	91:
		bTimer1															:= TRUE;
		IF tonTimer1.Q THEN
			bTimer1														:= FALSE;
			i4Step														:= 99;
		END_IF
		
	98:																														// Utility error hold - cleared by P_M01
		i4Step															:= 98;
		
	99:
		bRepressurizationDone											:= TRUE;
//		IF NOT bMultiProcess THEN
		Steam_Service_Req												:= FALSE;
//		END_IF
		Current_Step													:= 0;
		i4Step															:= 0;
	
END_CASE

IF i4Step > 0 AND i4Step < 80 THEN
	IF bMultiProcess THEN
		IF U.safe_shutdown_error_1 <> '' AND giSafeShutdown1RS = 0 THEN
			sSafeShutdownError1											:= U.safe_shutdown_error_1;
			giSafeShutdown1RS											:= RS_Number;
		ELSIF U.safe_shutdown_error_2 <> '' AND giSafeShutdown23RS = 0 THEN
			sSafeShutdownError2											:= U.safe_shutdown_error_2;
			giSafeShutdown23RS											:= RS_Number;
		ELSIF (giEvacuationErrorRS + giDesorptionErrorRS + giSafeShutdown1RS + giSafeShutdown23RS) > 0 THEN
			Cancel_Reactor_Set											:= TRUE;
		ELSIF U.os_air_unsafe_temp THEN
			Stop_Reactor_Set											:= TRUE;
		END_IF
	END_IF
	iStep																:= i4Step;
	Current_Step														:= iStep;
	A_Check_Process();
	i4Step																:= iStep;
END_IF
END_ACTION

ACTION A5_Adsorption:
// Phase 0 - FB_Reactor_Set.A5_Adsorption
// Rev 1.0 - May 13, 2024

CASE i5Step OF
	
	0:	;
		
	1:
		Cycle_Stage														:= 'adsorption.initialize';							// 2.d
		iRestartStep													:= 1;
		rTime2															:= m01.SP_adsorption_duration;						// 12
		IF R_S.reactor_pressure_error <> '' THEN
			sReactorError												:= R_S.reactor_pressure_error;
			sMessage													:= gsProcessCannotRun;
		ELSIF R_S.inlet_air_high_temp_count > _INLET_AIR_MAX_COUNT THEN
			sReactorError												:= F_Concat3(INT_TO_STRING(R_S.inlet_air_high_temp_count), ' ', gsSorbentTemperatureError);
			sMessage													:= gsProcessCannotRun;
		ELSE
			i5Step														:= i5Step + 1;
		END_IF
			
	2:
		IF NOT bMultiProcess THEN
			IF R_S.average_reactor_pressure_within_ambient THEN																// 2.c
				sReactorError											:= gsReactorsAtAmbientPressure;
				sMessage												:= gsProcessComplete;
			ELSIF NOT R_S.all_clamps_retracted THEN																			// 2.a
				sReactorError											:= gsDoorClampsExtendedError;
				sMessage												:= gsProcessCannotRun;
			ELSIF u.os_air_unsafe_temp THEN																					// 2.b
				sReactorError											:= gsOutsideTempRangeError;
				sMessage												:= gsProcessCannotRun;
			ELSE
				i5Step													:= i5Step + 1;
			END_IF
		ELSE
			i5Step														:= i5Step + 1;
		END_IF

	3:
		bTimer2															:= TRUE;											// 4
		IF R_S.r1_inlet_co2 < m01.SP_minimum_desired_inlet_co2_concentration_during_adsorption THEN							// 5.a
			sError														:= gsAdsorptionInletCo2LowError;
			sMessage													:= gsAdsorptionCo2LowCheck;
		END_IF
		R_S.close_all_valves											:= TRUE;											// 5.b
		U.drainage_on													:= TRUE;											// 5.d
		R_S.fan_vfd_percent												:= 0;												// 5.e
		rTime1															:= _VALVE_TIME;
		i5Step															:= i5Step + 1;
		
	4:
		bTimer1															:= TRUE;
		IF R_S.valves_clear THEN
			bTimer1														:= FALSE;
			i5Step														:= i5Step + 1;
		ELSIF tonTimer1.Q THEN
			bTimer1														:= FALSE;
			sReactorError												:= SEL(R_S.steam_control_valve_closed, gsSteamControlValveError, '');
			sReactorError												:= SEL(R_S.dead_air_valve_clear, gsDeadAirValveError, sReactorError);
			sReactorError												:= SEL(R_S.purge_valve_clear, gsPurgeValveError, sReactorError);
			sReactorError												:= SEL(R_S.cooling_valve_clear, gsCoolingValveError, sReactorError);
			sReactorError												:= SEL(R_S.steam_header_valve_clear, gsSteamHeaderValveError, sReactorError);
			sMessage													:= gsReactorSetCannotRun;
		END_IF

	5:
		R_S.open_repres_valves											:= TRUE;											// 6
		rTime1															:= _VALVE_TIME;
		i5Step															:= i5Step + 1;

	6:
		bTimer1															:= TRUE;
		IF R_S.repres_valve_error = '' THEN
			bTimer1														:= FALSE;
			R_S.co2_outside_sensors_on									:= TRUE;											// 7
			R_S.open_all_doors											:= TRUE;											// 8
			Cycle_Stage													:= 'adsorption.open_doors';							// 8.a
			rTime1														:= m01.SP_doorsopenclose_timedelay * _MINUTES;		// 8.b
			i5Step														:= i5Step + 1;
		ELSIF tonTimer1.Q THEN
			bTimer1														:= FALSE;
			sReactorError												:= R_S.repres_valve_error;
			sMessage													:= gsProcessCannotRun;
		END_IF
							
	7:
		bTimer1															:= TRUE;
		IF R_S.all_doors_open THEN
			bTimer1														:= FALSE;
			R_S.fan_vfd_percent											:= Fan_setpoint;									// 9
			Cycle_Stage													:= 'adsorption.turn_on_fans';						// 9.a
			rSP1														:= m01.SP_unacceptable_duration_from_adsorption_start_until_sorbent_cool * _MINUTES;	// 10.c
			rSP2														:= m01.SP_undesirable_duration_from_adsorption_start_until_sorbent_cool * _MINUTES;		// 10.b
			rSP3														:= m01.SP_target_duration_from_adsorption_start_until_sorbent_cool * _MINUTES;			// 10.a
			i5Step														:= i5Step + 1;
		ELSIF tonTimer1.Q THEN
			bTimer1														:= FALSE;
			sReactorError												:= gsDoorsNotOpenError;
			sMessage													:= gsProcessCannotRun;
		END_IF
		
	8:
		rTime															:= TIME_TO_REAL(tonTimer2.ET);
		IF rTime >= rSP1 THEN																								// 10.c
			IF R_S.inlet_air_high_temp_count = 0 THEN																		// 10.c.i
				sPauseError												:= gsAdsorptionUnacceptableTimeError;
				sMessage												:= gsReactorSetWillPause;												
			ELSE
				sSafeShutdownError1										:= gsAdsorptionTimeOutError;						// 10.c.ii - Safe Shutdown 1
			END_IF
		ELSIF rTime >= rSP2 THEN																							// 10.b
			IF R_S.inlet_air_high_temp_count = 0 THEN
				sError													:= gsAdsorptionAcceptableButNotIdealTimeError;																
				i5Step													:= i5Step + 1;
			END_IF
		ELSIF rTime >= rSP3 THEN																							// 10.c
			IF R_S.inlet_air_high_temp_count = 0 THEN																	
				i5Step													:= i5Step + 1;
			END_IF
		END_IF

	9:
		R_S.co2_inside_sensors_on										:= TRUE;											// 11
		Cycle_Stage														:= 'adsorption.adsorption';							// 11.a
		i5Step 															:= i5Step + 1;
		
	10:
		IF tonTimer2.Q THEN																									// 12
			bTimer2														:= FALSE;
			R_S.fan_vfd_percent											:= 0;
			Cycle_Stage													:= 'adsorption.turn_off_fans';						// 12.a
			rTime1														:= _FAN_SHUTDOWN_TIME;
			i5Step														:= i5Step + 1;
		END_IF

	11:
		bTimer1															:= TRUE;
		IF tonTimer1.Q THEN
			bTimer1														:= FALSE;	
			R_S.close_all_doors											:= TRUE;											// 13
			Cycle_Stage													:= 'adsorption.close_doors';						// 13.a
			rTime1														:= m01.SP_doorsopenclose_timedelay * _MINUTES;										// 13.b
			i5Step														:= i5Step + 1;
		END_IF
		
	12:
		bTimer1															:= TRUE;
		IF tonTimer1.Q THEN
			bTimer1														:= FALSE;
			R_S.co2_sensors_off											:= TRUE;											// 14
			rTime1														:= m01.SP_dead_time_in_cycle_duration;				// 15
			Cycle_Stage													:= 'adsorption.cycle_dead_time';					// 15.a
			i5Step														:= i5Step + 1;
		END_IF
		
	13:
		bTimer1															:= TRUE;
		IF tonTimer1.Q THEN
			bTimer1														:= FALSE;
			i5Step														:= 99;
		END_IF
				
	80:																														// Manual process closing
		Cycle_Stage														:= 'adsorption.stopping';
		R_S.fan_vfd_percent												:= 0;
		R_S.co2_sensors_off												:= TRUE;
		R_S.close_repres_valves											:= TRUE;
		rTime1															:= _STOPPING_TIME;
		i5Step															:= i5Step + 1;
		
	81:
		bTimer1															:= TRUE;
		IF tonTimer1.Q THEN
			bTimer1														:= FALSE;
			i5Step														:= 99;
		END_IF
		
	90:																														// Automatic process stopping
		Cycle_Stage														:= 'adsorption.stopping';
		R_S.fan_vfd_percent												:= 0;
		R_S.co2_sensors_off												:= TRUE;
		R_S.close_repres_valves											:= TRUE;
		rTime1															:= _STOPPING_TIME;
		i5Step															:= i5Step + 1;
		
	91:
		bTimer1															:= TRUE;
		IF tonTimer1.Q THEN
			bTimer1														:= FALSE;
			i5Step														:= 99;
		END_IF
		
	98:																														// Utility error hold - cleared by P_M01
		i5Step															:= 98;
		
	99:
		bAdsorptionDone													:= TRUE;
		bTimer2															:= FALSE;
		U.drainage_on													:= FALSE;
		Current_Step													:= 0;
		i5Step															:= 0;
	
END_CASE

IF i5Step > 0 AND i5Step < 80 THEN
	IF bMultiProcess THEN
		IF U.safe_shutdown_error_1 <> '' AND giSafeShutdown1RS = 0 THEN
			sSafeShutdownError1											:= U.safe_shutdown_error_1;
			giSafeShutdown1RS											:= RS_Number;
		ELSIF U.safe_shutdown_error_2 <> '' AND giSafeShutdown23RS = 0 THEN
			sSafeShutdownError2											:= U.safe_shutdown_error_2;
			giSafeShutdown23RS											:= RS_Number;
		ELSIF sSafeShutdownError1 <> '' AND giSafeShutdown1RS = 0 THEN
			giSafeShutdown1RS											:= RS_Number;
		ELSIF (giEvacuationErrorRS + giDesorptionErrorRS + giSafeShutdown1RS + giSafeShutdown23RS) > 0 THEN
			Cancel_Reactor_Set											:= TRUE;
		ELSIF U.os_air_unsafe_temp THEN
			Stop_Reactor_Set											:= TRUE;
		END_IF
	END_IF
	iStep																:= i5Step;
	Current_Step														:= iStep;
	A_Check_Process();
	i5Step																:= iStep;
END_IF
END_ACTION

ACTION A5_Adsorption_Test:
// Phase 0 - FB_Reactor_Set.A5_Adsorption_Test
// Rev 1.0 - June 3, 2024

CASE i5Step OF	

	0:	;
		
	1:
		Cycle_Stage														:= 'adsorption.initialize';							// 2.d
		//iRestartStep													:= 1;
		rTime2															:= m01.SP_adsorption_duration * _MINUTES;			// 12
		IF R_S.reactor_pressure_error <> '' THEN
			sReactorError												:= R_S.reactor_pressure_error;
			sMessage													:= gsProcessCannotRun;
		ELSE
			R_S.retract_all_clamps 										:= TRUE;
			rTime1														:= m01.SP_clampsretract_timedelay;
			i5Step														:= i5Step + 1;
		END_IF
			
	2:
		IF NOT bMultiProcess THEN
			IF R_S.average_reactor_pressure_within_ambient THEN																// 2.c
				sReactorError											:= gsReactorsAtAmbientPressure;
				sMessage												:= gsProcessComplete;
			ELSE
				i5Step													:= i5Step + 1;
			END_IF
		ELSE
			i5Step														:= i5Step + 1;
		END_IF

	3:
		bTimer1															:= TRUE;
		IF R_S.all_clamps_retracted THEN																					// 2.a
			bTimer1														:= FALSE;
			i5Step														:= i5Step + 1;
		ELSE
			sReactorError												:= gsDoorClampsExtendedError;
			sMessage													:= gsProcessCannotRun;
		END_IF
		
	4:
		R_S.close_all_valves											:= TRUE;											// 5.b
		U.drainage_on													:= TRUE;											// 5.d
		R_S.fan_vfd_percent												:= 0;												// 5.e
		rTime1															:= _VALVE_TIME;
		i5Step															:= i5Step + 1;
		
	5:
		bTimer1															:= TRUE;
		IF R_S.valves_clear THEN
			bTimer1														:= FALSE;
			i5Step														:= i5Step + 2;
		ELSIF tonTimer1.Q THEN
			bTimer1														:= FALSE;
			sReactorError												:= SEL(R_S.steam_control_valve_closed, gsSteamControlValveError, '');
			sReactorError												:= SEL(R_S.dead_air_valve_clear, gsDeadAirValveError, sReactorError);
			sReactorError												:= SEL(R_S.purge_valve_clear, gsPurgeValveError, sReactorError);
			sReactorError												:= SEL(R_S.cooling_valve_clear, gsCoolingValveError, sReactorError);
			sReactorError												:= SEL(R_S.steam_header_valve_clear, gsSteamHeaderValveError, sReactorError);
			sMessage													:= gsReactorSetCannotRun;
		END_IF

	6:
		R_S.open_repres_valves											:= TRUE;											// 6
		rTime1															:= _VALVE_TIME;
		i5Step															:= i5Step + 1;

	7:
		bTimer1															:= TRUE;
		IF R_S.repres_valve_error = '' THEN
			bTimer1														:= FALSE;
			R_S.co2_inside_sensors_on									:= TRUE;											// 7
			R_S.open_all_doors											:= TRUE;											// 8
			Cycle_Stage													:= 'adsorption.open_doors';							// 8.a
			rTime1														:= m01.SP_doorsopenclose_timedelay * _MINUTES;		// 8.b
			i5Step														:= i5Step + 1;
		ELSIF tonTimer1.Q THEN
			bTimer1														:= FALSE;
			sReactorError												:= R_S.repres_valve_error;
			sMessage													:= gsProcessCannotRun;
		END_IF
							
	8:
		bTimer1															:= TRUE;
		//IF R_S.all_doors_open THEN
		IF tonTimer1.Q THEN
			bTimer1														:= FALSE;
			R_S.close_repres_valves										:= TRUE;		
			R_S.fan_vfd_percent											:= Fan_setpoint;									// 9
			Cycle_Stage													:= 'adsorption.turn_on_fans';						// 9.a
		
			i5Step														:= i5Step + 1;
		END_IF
		
	9:
		IF R_S.sorbent_high_temp <=  m01.SP_adsorption_sorbent_hightemp_startco2analyzer THEN 
				i5Step														:= i5Step + 1;
		END_IF

	10:
		//R_S.co2_inside_sensors_on										:= TRUE;											// 11
		bTimer2															:= TRUE;	
		Cycle_Stage														:= 'adsorption.adsorption';							// 11.a
		IF R_S.R1_outlet_co2 >= m01.SP_adsorption_outletco2_highlimit AND tonTimer2.Q THEN
			bTimer2															:= FALSE;	
			i5Step 															:= i5Step + 1;
		END_IF
		
	11:
		
		R_S.fan_vfd_percent											:= 0;
		Cycle_Stage													:= 'adsorption.turn_off_fans';						// 12.a
		rTime1														:= _FAN_SHUTDOWN_TIME;
		i5Step														:= i5Step + 1;
	

	12:
		bTimer1															:= TRUE;
		IF tonTimer1.Q THEN
			bTimer1														:= FALSE;	
			R_S.close_all_doors											:= TRUE;											// 13
			Cycle_Stage													:= 'adsorption.close_doors';						// 13.a
			rTime1														:= m01.SP_doorsopenclose_timedelay * _MINUTES;										// 13.b
			i5Step														:= i5Step + 1;
		END_IF
		
	13:
		bTimer1															:= TRUE;
		IF tonTimer1.Q THEN
			bTimer1														:= FALSE;
			R_S.co2_sensors_off											:= TRUE;											// 14
			rTime1														:= m01.SP_dead_time_in_cycle_duration;				// 15
			Cycle_Stage													:= 'adsorption.cycle_dead_time';					// 15.a
			i5Step														:= i5Step + 1;
		END_IF
		
	14:
		bTimer1															:= TRUE;
		IF tonTimer1.Q THEN
			bTimer1														:= FALSE;
			i5Step														:= 99;
		END_IF
				
	80:																														// Manual process closing
		Cycle_Stage														:= 'adsorption.stopping';
		R_S.fan_vfd_percent												:= 0;
		R_S.co2_sensors_off												:= TRUE;
		R_S.close_repres_valves											:= TRUE;
		rTime1															:= _STOPPING_TIME;
		i5Step															:= i5Step + 1;
		
	81:
		bTimer1															:= TRUE;
		IF tonTimer1.Q THEN
			bTimer1														:= FALSE;
			i5Step														:= 99;
		END_IF
		
	90:																														// Automatic process stopping
		Cycle_Stage														:= 'adsorption.stopping';
		R_S.fan_vfd_percent												:= 0;
		R_S.co2_sensors_off												:= TRUE;
		R_S.close_repres_valves											:= TRUE;
		rTime1															:= _STOPPING_TIME;
		i5Step															:= i5Step + 1;
		
	91:
		bTimer1															:= TRUE;
		IF tonTimer1.Q THEN
			bTimer1														:= FALSE;
			i5Step														:= 99;
		END_IF
		
	98:																														// Utility error hold - cleared by P_M01
		i5Step															:= 98;
		
	99:
		bAdsorptionDone													:= TRUE;
		//bTimer2															:= FALSE;
		U.drainage_on													:= FALSE;
		Current_Step													:= 0;
		i5Step															:= 0;
	
END_CASE

IF i5Step > 0 AND i5Step < 80 THEN
	IF bMultiProcess THEN
		IF U.safe_shutdown_error_1 <> '' AND giSafeShutdown1RS = 0 THEN
			sSafeShutdownError1											:= U.safe_shutdown_error_1;
			giSafeShutdown1RS											:= RS_Number;
		ELSIF U.safe_shutdown_error_2 <> '' AND giSafeShutdown23RS = 0 THEN
			sSafeShutdownError2											:= U.safe_shutdown_error_2;
			giSafeShutdown23RS											:= RS_Number;
		ELSIF sSafeShutdownError1 <> '' AND giSafeShutdown1RS = 0 THEN
			giSafeShutdown1RS											:= RS_Number;
		ELSIF (giEvacuationErrorRS + giDesorptionErrorRS + giSafeShutdown1RS + giSafeShutdown23RS) > 0 THEN
			Cancel_Reactor_Set											:= TRUE;
		ELSIF U.os_air_unsafe_temp THEN
			Stop_Reactor_Set											:= TRUE;
		END_IF
	END_IF
	iStep																:= i5Step;
	Current_Step														:= iStep;
	A_Check_Process();
	i5Step																:= iStep;
END_IF
END_ACTION

ACTION A5_Adsorption_Test_Auto:
// Phase 0 - FB_Reactor_Set.A5_Adsorption_Test
// Rev 1.0 - June 3, 2024

CASE i5Step OF	

	0:	;
		
	1:
		Cycle_Stage														:= 'adsorption.initialize';							// 2.d
		//iRestartStep													:= 1;
		rTime1														:= 5 * _SECONDS;
		i5Step														:= i5Step + 1;
		
			
	2:
		bTimer1 := TRUE;
		IF sita_bits[3].1 THEN 
			bTimer1 := FALSE;
			i5Step := 90;
		ELSIF tonTimer1.Q AND  sita_bits[3].2 THEN 
			bTimer1														:= FALSE;
			sReactorError												:= 'Adsorption Error';
			sMessage													:= 'Auto Test';
		END_IF

	
	80:																														// Manual process closing
		Cycle_Stage														:= 'adsorption.stopping';
		rTime1															:= _STOPPING_TIME;
		i5Step															:= i5Step + 1;
		
	81:
		bTimer1															:= TRUE;
		IF tonTimer1.Q THEN
			bTimer1														:= FALSE;
			i5Step														:= 99;
		END_IF
		
	90:																														// Automatic process stopping
		Cycle_Stage														:= 'adsorption.stopping';
		rTime1															:= _STOPPING_TIME;
		i5Step															:= i5Step + 1;
		
	91:
		bTimer1															:= TRUE;
		IF tonTimer1.Q THEN
			bTimer1														:= FALSE;
			i5Step														:= 99;
		END_IF
		
	98:																														// Utility error hold - cleared by P_M01
		i5Step															:= 98;
		
	99:
		bAdsorptionDone													:= TRUE;
		//bTimer2															:= FALSE;
		U.drainage_on													:= FALSE;
		Current_Step													:= 0;
		i5Step															:= 0;
	
END_CASE

IF i5Step > 0 AND i5Step < 80 THEN
	IF bMultiProcess THEN
		IF U.safe_shutdown_error_1 <> '' AND giSafeShutdown1RS = 0 THEN
			sSafeShutdownError1											:= U.safe_shutdown_error_1;
			giSafeShutdown1RS											:= RS_Number;
		ELSIF U.safe_shutdown_error_2 <> '' AND giSafeShutdown23RS = 0 THEN
			sSafeShutdownError2											:= U.safe_shutdown_error_2;
			giSafeShutdown23RS											:= RS_Number;
		ELSIF sSafeShutdownError1 <> '' AND giSafeShutdown1RS = 0 THEN
			giSafeShutdown1RS											:= RS_Number;
		ELSIF (giEvacuationErrorRS + giDesorptionErrorRS + giSafeShutdown1RS + giSafeShutdown23RS) > 0 THEN
			Cancel_Reactor_Set											:= TRUE;
		ELSIF U.os_air_unsafe_temp THEN
			Stop_Reactor_Set											:= TRUE;
		END_IF
	END_IF
	iStep																:= i5Step;
	Current_Step														:= iStep;
	A_Check_Process();
	i5Step																:= iStep;
END_IF
END_ACTION

ACTION A6_Evacuation:
// Phase 0 - FB_State_Machine.A6_Evacuation
// Rev 1.0 - May 13, 2024

CASE i6Step OF
	
	0:	;
	
	1:
		Cycle_Stage														:= 'evacuation.initialize';							// 1.a
		iRestartStep													:= 1;
		rTime2															:= m01.SP_evacuation_duration;
		IF U.utility_error <> '' THEN																						// 2
			sUtilityError												:= U.utility_error;
			sMessage													:= gsSystemCannotRun;
		ELSIF R_S.reactor_pressure_error <> '' THEN
			sReactorError												:= R_S.reactor_pressure_error;
			sMessage													:= gsReactorSetCannotRun;
		ELSE
			R_S.close_all_doors											:= TRUE;
			rTime1														:= m01.SP_doorsopenclose_timedelay * _MINUTES;
			i6Step														:= i6Step + 1;
		END_IF
		
	2:
		bTimer1															:= TRUE;
		IF R_S.all_doors_closed THEN																						// 1.c.ii
			bTimer1														:= FALSE;
			R_S.close_all_valves										:= TRUE;											// 4.a
			rTime1														:= _VALVE_TIME; 
			i6Step														:= i6Step + 1;
		ELSIF tonTimer1.Q THEN
			bTimer1														:= FALSE;
			sReactorError												:= gsDoorsNotClosedError;
			sMessage													:= gsReactorSetCannotRun;
		END_IF

	3:
		bTimer1															:= TRUE;
		bTimer2															:= TRUE;											// 3
		IF R_S.valves_clear THEN
			bTimer1														:= FALSE;
			U.product_vacuum_backfeed_valve								:= _OPEN;											// 4.a.ii
			rTime1														:= _VALVE_TIME; 
			i6Step														:= i6Step + 1;
		ELSIF tonTimer1.Q THEN
			bTimer1														:= FALSE;
			sReactorError												:= SEL(R_S.steam_control_valve_closed, gsSteamControlValveError, '');
			sReactorError												:= SEL(R_S.dead_air_valve_clear, gsDeadAirValveError, sReactorError);
			sReactorError												:= SEL(R_S.purge_valve_clear, gsPurgeValveError, sReactorError);
			sReactorError												:= SEL(R_S.cooling_valve_clear, gsCoolingValveError, sReactorError);
			sReactorError												:= SEL(R_S.steam_header_valve_clear, gsSteamHeaderValveError, sReactorError);
			sMessage													:= gsReactorSetCannotRun;
		END_IF

	4:
		bTimer1															:= TRUE;
		IF U.product_vacuum_backfeed_valve_open THEN
			bTimer1														:= FALSE;
			U.drainage_on												:= TRUE;											// 4.c
			R_S.co2_outside_sensors_on									:= TRUE;											// 5
			R_S.close_repres_valves										:= TRUE;											// 6
			rTime1														:= _VALVE_TIME; 
			i6Step														:= i6Step + 1;
		ELSIF tonTimer1.Q THEN
			bTimer1														:= FALSE;
			sUtilityError												:= gsProductVacuumBackfeedValveError;
			sMessage													:= gsSystemCannotRun;
		END_IF
			
	5:		
		bTimer1															:= TRUE;	
		IF R_S.repres_valve_error = '' THEN
			bTimer1														:= FALSE;
			R_S.extend_all_clamps										:= TRUE;											// 7
			U.dead_air_vacuum_pump										:= TRUE;											// 8
			Cycle_Stage													:= 'evacuation.evacuate_lines';						// 8.a
			i6Step														:= i6Step + 1;
		ELSIF tonTimer1.Q THEN
			bTimer1														:= FALSE;
			sReactorError												:= R_S.repres_valve_error;
			sMessage													:= gsProcessCannotRun;
		END_IF
		
	6:
		IF U.dead_air_line_pres < m01.SP_evacuation_unacceptable_pressure THEN												// 9
			R_S.dead_air_valve											:= TRUE;											// 9.a
			Cycle_Stage													:= 'evacuation.evacuation';							// 10
			i6Step														:= i6Step + 1;			
		ELSIF tonTimer2.Q OR U.dead_air_line_pres_error THEN																// 9.b
			bTimer2														:= FALSE;
			sReactorError												:= gsUnableToEvacuateLinesError;					// Raise error & stop reactor set				
			sMessage													:= gsSystemWillStop;
			bEvacuationRSError											:= TRUE;											// Stop evacuation for all reactor sets in evacuation. Allow other reactor sets to complete their current cycle.
		END_IF
		 
	7:
		IF tonTimer2.Q THEN																									// 11
			bTimer2														:= FALSE;											// 14
			iStatus														:= F_LowMidHigh(R_S.average_reactor_pressure, m01.SP_evacuation_ideal_pressure, m01.SP_evacuation_unacceptable_pressure, 0);
			IF iStatus = eLow THEN																							// 11.a
				i6Step													:= i6Step + 1;
			ELSIF iStatus = eMid THEN																						// 11.b
				sError													:= gsVacuumPressureAcceptableBotNotIdealError;
				sMessage												:= gsProcessWillContinue;
				i6Step													:= i6Step + 1;
			ELSE																											// 11.c
				sReactorError											:= gsInsufficientVacuumPressureError;
				sMessage												:= gsReactorSetWillPause;
			END_IF
		END_IF
	
	8:
		R_S.dead_air_valve												:= FALSE;											// 12
		U.dead_air_vacuum_pump											:= FALSE;											// 13
		IF R_S.all_clamps_extended THEN																						// 15
			i6Step														:= i6Step + 1;
		ELSE
			sReactorError												:= gsClampExtendError;
			sMessage													:= gsProcessCannotContinue;
		END_IF

	9:
		Cycle_Stage														:= 'evacuation.leak_check';							// 16
		rTime2															:= m01.SP_leak_test_duration;						// 17
		rR1SavedPressure												:= R_S.R1_reactor_pres;
		rR2SavedPressure												:= R_S.R2_reactor_pres;
		rR3SavedPressure												:= R_S.R3_reactor_pres;
		rR4SavedPressure												:= R_S.R4_reactor_pres;
		i6Step															:= i6Step + 1;

	10:
		bTimer2															:= TRUE;
		IF tonTimer2.Q THEN																									// 18
			bTimer2														:= FALSE;
			rR1SavedPressure											:= R_S.R1_reactor_pres - rR1SavedPressure;
			rR2SavedPressure											:= R_S.R2_reactor_pres - rR2SavedPressure;
			rR3SavedPressure											:= R_S.R3_reactor_pres - rR3SavedPressure;
			rR4SavedPressure											:= R_S.R4_reactor_pres - rR4SavedPressure;
			rSP1														:= m01.SP_target_pressure_change;
			rSP2														:= m01.SP_unacceptable_pressure_change;
			iR1Leakage													:= F_LowMidHigh(rR1SavedPressure, rSP1, rSP2, 0);
			iR2Leakage													:= F_LowMidHigh(rR2SavedPressure, rSP1, rSP2, 0);
			iR3Leakage													:= F_LowMidHigh(rR3SavedPressure, rSP1, rSP2, 0);
			iR4Leakage													:= F_LowMidHigh(rR4SavedPressure, rSP1, rSP2, 0);
			sLeakageAcceptable											:= SEL(iR1Leakage = 1, '', 'R1 ');
			sLeakageAcceptable											:= SEL(iR2Leakage = 1, sLeakageAcceptable, CONCAT(sLeakageAcceptable, 'R2 '));
			sLeakageAcceptable											:= SEL(iR3Leakage = 1, sLeakageAcceptable, CONCAT(sLeakageAcceptable, 'R3 '));
			sLeakageAcceptable											:= SEL(iR4Leakage = 1, sLeakageAcceptable, CONCAT(sLeakageAcceptable, 'R4 '));
			sLeakageUnacceptable										:= SEL(iR1Leakage = 2, '', 'R1 ');
			sLeakageUnacceptable										:= SEL(iR2Leakage = 2, sLeakageUnacceptable, CONCAT(sLeakageUnacceptable, 'R2 '));
			sLeakageUnacceptable										:= SEL(iR3Leakage = 2, sLeakageUnacceptable, CONCAT(sLeakageUnacceptable, 'R3 '));
			sLeakageUnacceptable										:= SEL(iR4Leakage = 2, sLeakageUnacceptable, CONCAT(sLeakageUnacceptable, 'R4 '));
			IF sLeakageUnacceptable = '' THEN
				R_S.vacuum_holding										:= TRUE;											// 18.a.i
				R_S.co2_sensors_off										:= TRUE;											// 19
				IF sLeakageAcceptable <> '' THEN
					sError												:= CONCAT(sLeakageAcceptable, gsVacuumPressureAcceptableBotNotIdealError);		// 18.b.i
					sMessage											:= gsReactorSetWillContinue;
				END_IF																										// else 18.a
				i6Step													:= 99;
			ELSE
				R_S.vacuum_holding										:= FALSE;											// 18.c.ii
				sReactorError											:= CONCAT(sLeakageUnacceptable, gsVacuumPressureUnacceptableError);				// 18.c.i
				sMessage												:= gsReactorSetWillPause;
			END_IF
		END_IF			
		
	80:																														// Stop process
		Cycle_Stage														:= 'evacuation.stopping';
		R_S.co2_sensors_off												:= TRUE;
		R_S.dead_air_valve												:= FALSE;
		U.dead_air_vacuum_pump											:= FALSE;
		U.product_vacuum_backfeed_valve									:= _CLOSED;
		rTime1															:= _STOPPING_TIME;
		i6Step															:= i6Step + 1;
		
	81:
		bTimer1															:= TRUE;
		IF tonTimer1.Q THEN
			bTimer1														:= FALSE;
			i6Step														:= 99;
		END_IF

	90:																														// Automatic process stopping
		Cycle_Stage														:= 'evacuation.stopping';
		R_S.co2_sensors_off												:= TRUE;
		R_S.dead_air_valve												:= FALSE;
		U.dead_air_vacuum_pump											:= FALSE;
		U.product_vacuum_backfeed_valve									:= _CLOSED;
		rTime1															:= _STOPPING_TIME;
		i6Step															:= i6Step + 1;
		
	91:
		bTimer1															:= TRUE;
		IF tonTimer1.Q THEN
			bTimer1														:= FALSE;
			i6Step														:= 99;
		END_IF
		
	98:																														// Utility error hold - cleared by P_M01
		i6Step															:= 98;
		
	99:
		IF bStopAfterEvacuation THEN
			bStop														:= TRUE;
			Stop_M01_RS													:= TRUE;											// Stop Reactor in P_M01.A_AutoMode
			bStopAfterEvacuation										:= FALSE;
		END_IF
		bEvacuationDone													:= TRUE;
		U.drainage_on													:= FALSE;
		Current_Step													:= 0;
		i6Step															:= 0;
	
END_CASE

IF i6Step > 0 AND i6Step < 80 THEN
	IF bMultiProcess THEN
		IF U.safe_shutdown_error_1 <> '' AND giSafeShutdown1RS = 0 THEN
			sSafeShutdownError1											:= U.safe_shutdown_error_1;
			giSafeShutdown1RS											:= RS_Number;
		ELSIF U.safe_shutdown_error_2 <> '' AND giSafeShutdown23RS = 0 THEN
			sSafeShutdownError2											:= U.safe_shutdown_error_2;
			giSafeShutdown23RS											:= RS_Number;
		ELSIF bEvacuationRSError AND giEvacuationErrorRS = 0 THEN															// Error occured in this reactor set
			bEvacuationRSError											:= FALSE;
			giEvacuationErrorRS											:= RS_Number;										// Save reactor set number to handle error in other reactor sets
		ELSIF giDesorptionErrorRS > 0 THEN
			bStopAfterEvacuation										:= TRUE;
		ELSIF U.os_air_unsafe_temp OR (giEvacuationErrorRS + giSafeShutdown1RS + giSafeShutdown23RS) > 0 THEN 
			Stop_Reactor_Set											:= TRUE;
		END_IF
	END_IF
	iStep																:= i6Step;
	Current_Step														:= iStep;
	A_Check_Process();
	i6Step																:= iStep;
END_IF
END_ACTION

ACTION A6_Evacuation_Test:
// Phase 0 - FB_State_Machine.A6_Evacuation_Test
// Rev 1.0 - June 3, 2024

CASE i6Step OF
	
	0:	;
	
	1:
		Cycle_Stage														:= 'evacuation.initialize';							// 1.a
		iRestartStep													:= 1;
		rTime2															:= m01.SP_evacuation_duration;
		IF U.utility_error <> '' THEN																						// 2
			sUtilityError												:= U.utility_error;
			sMessage													:= gsSystemCannotRun;
		ELSIF R_S.reactor_pressure_error <> '' THEN
			sReactorError												:= R_S.reactor_pressure_error;
			sMessage													:= gsReactorSetCannotRun;
		ELSE
			R_S.close_all_doors											:= TRUE;
			rTime1														:= m01.SP_doorsopenclose_timedelay * _MINUTES;
			i6Step														:= i6Step + 1;
		END_IF
		
	2:
		bTimer1															:= TRUE;
		//IF R_S.all_doors_closed THEN
		IF NOT R_S.all_doors_open THEN																						// 1.c.ii
			bTimer1														:= FALSE;
			R_S.close_all_valves										:= TRUE;											// 4.a
			rTime1														:= _VALVE_TIME; 
			i6Step														:= i6Step + 1;
		ELSIF tonTimer1.Q THEN
			bTimer1														:= FALSE;
			sReactorError												:= gsDoorsNotClosedError;
			sMessage													:= gsReactorSetCannotRun;
		END_IF

	3:
		bTimer1															:= TRUE;
		bTimer2															:= TRUE;											// 3
		IF R_S.valves_clear THEN
			bTimer1														:= FALSE;
			//U.product_vacuum_backfeed_valve								:= _OPEN;											// 4.a.ii
			//rTime1														:= _VALVE_TIME; 
			i6Step														:= i6Step + 1;
		ELSIF tonTimer1.Q THEN
			bTimer1														:= FALSE;
			sReactorError												:= SEL(R_S.steam_control_valve_closed, gsSteamControlValveError, '');
			sReactorError												:= SEL(R_S.dead_air_valve_clear, gsDeadAirValveError, sReactorError);
			sReactorError												:= SEL(R_S.purge_valve_clear, gsPurgeValveError, sReactorError);
			sReactorError												:= SEL(R_S.cooling_valve_clear, gsCoolingValveError, sReactorError);
			sReactorError												:= SEL(R_S.steam_header_valve_clear, gsSteamHeaderValveError, sReactorError);
			sMessage													:= gsReactorSetCannotRun;
		END_IF

	4:
		//bTimer1															:= TRUE;
		//IF U.product_vacuum_backfeed_valve_open THEN
			//bTimer1														:= FALSE;
			//U.drainage_on												:= TRUE;											// 4.c
			R_S.co2_outside_sensors_on									:= TRUE;											// 5
			R_S.close_repres_valves										:= TRUE;											// 6
			rTime1														:= _VALVE_TIME; 
			i6Step														:= i6Step + 1;
		//ELSIF tonTimer1.Q THEN
			//bTimer1														:= FALSE;
			//sUtilityError												:= gsSystemCannotRun;
		//END_IF
			
	5:		
		bTimer1															:= TRUE;	
		IF R_S.repres_valve_error = '' THEN
			bTimer1														:= FALSE;
			R_S.extend_all_clamps										:= TRUE;											// 7
			U.dead_air_vacuum_pump										:= TRUE;											// 8
			R_S.dead_air_valve											:= TRUE;											// 9.a
			Cycle_Stage													:= 'evacuation.evacuation';							// 10
//			Cycle_Stage													:= 'evacuation.evacuate_lines';						// 8.a
			i6Step														:= i6Step + 1;
		ELSIF tonTimer1.Q THEN
			bTimer1														:= FALSE;
			sReactorError												:= R_S.repres_valve_error;
			sMessage													:= gsProcessCannotRun;
		END_IF
		
	6:
		IF U.dead_air_line_pres <= m01.SP_evacuation_unacceptable_pressure THEN												// 9
			i6Step														:= i6Step + 2;			
		//ELSIF tonTimer2.Q OR U.dead_air_line_pres_error THEN
		ELSIF U.dead_air_line_pres_error THEN																// 9.b
			bTimer2														:= FALSE;
			sReactorError												:= gsUnableToEvacuateLinesError;					// Raise error & stop reactor set				
			sMessage													:= gsSystemWillStop;
			bEvacuationRSError											:= TRUE;											// Stop evacuation for all reactor sets in evacuation. Allow other reactor sets to complete their current cycle.
		END_IF
		 
	7:
		IF tonTimer2.Q THEN																									// 11
			bTimer2														:= FALSE;											// 14
			iStatus														:= F_LowMidHigh(R_S.average_reactor_pressure, m01.SP_evacuation_ideal_pressure, m01.SP_evacuation_unacceptable_pressure, 0);
			IF iStatus = eLow THEN																							// 11.a
				i6Step													:= i6Step + 1;
			ELSIF iStatus = eMid THEN																						// 11.b
				sError													:= gsVacuumPressureAcceptableBotNotIdealError;
				sMessage												:= gsProcessWillContinue;
				i6Step													:= i6Step + 1;
			ELSE																											// 11.c
				sReactorError											:= gsInsufficientVacuumPressureError;
				sMessage												:= gsReactorSetWillPause;
			END_IF
		END_IF
	
	8:
		R_S.dead_air_valve												:= FALSE;											// 12
		U.dead_air_vacuum_pump											:= FALSE;											// 13
		i6Step															:= 99;
//		IF R_S.all_clamps_extended THEN																						// 15
//			i6Step														:= 99;
//		ELSE
//			sReactorError												:= gsClampExtendError;
//			sMessage													:= gsProcessCannotContinue;
//		END_IF

	9:
		Cycle_Stage														:= 'evacuation.leak_check';							// 16
		rTime2															:= m01.SP_leak_test_duration;						// 17
		rR1SavedPressure												:= R_S.R1_reactor_pres;
		rR2SavedPressure												:= R_S.R2_reactor_pres;
		rR3SavedPressure												:= R_S.R3_reactor_pres;
		rR4SavedPressure												:= R_S.R4_reactor_pres;
		i6Step															:= i6Step + 1;

	10:
		bTimer2															:= TRUE;
		IF tonTimer2.Q THEN																									// 18
			bTimer2														:= FALSE;
			rR1SavedPressure											:= R_S.R1_reactor_pres - rR1SavedPressure;
			rR2SavedPressure											:= R_S.R2_reactor_pres - rR2SavedPressure;
			rR3SavedPressure											:= R_S.R3_reactor_pres - rR3SavedPressure;
			rR4SavedPressure											:= R_S.R4_reactor_pres - rR4SavedPressure;
			rSP1														:= m01.SP_target_pressure_change;
			rSP2														:= m01.SP_unacceptable_pressure_change;
			iR1Leakage													:= F_LowMidHigh(rR1SavedPressure, rSP1, rSP2, 0);
			iR2Leakage													:= F_LowMidHigh(rR2SavedPressure, rSP1, rSP2, 0);
			iR3Leakage													:= F_LowMidHigh(rR3SavedPressure, rSP1, rSP2, 0);
			iR4Leakage													:= F_LowMidHigh(rR4SavedPressure, rSP1, rSP2, 0);
			sLeakageAcceptable											:= SEL(iR1Leakage = 1, '', 'R1 ');
			sLeakageAcceptable											:= SEL(iR2Leakage = 1, sLeakageAcceptable, CONCAT(sLeakageAcceptable, 'R2 '));
			sLeakageAcceptable											:= SEL(iR3Leakage = 1, sLeakageAcceptable, CONCAT(sLeakageAcceptable, 'R3 '));
			sLeakageAcceptable											:= SEL(iR4Leakage = 1, sLeakageAcceptable, CONCAT(sLeakageAcceptable, 'R4 '));
			sLeakageUnacceptable										:= SEL(iR1Leakage = 2, '', 'R1 ');
			sLeakageUnacceptable										:= SEL(iR2Leakage = 2, sLeakageUnacceptable, CONCAT(sLeakageUnacceptable, 'R2 '));
			sLeakageUnacceptable										:= SEL(iR3Leakage = 2, sLeakageUnacceptable, CONCAT(sLeakageUnacceptable, 'R3 '));
			sLeakageUnacceptable										:= SEL(iR4Leakage = 2, sLeakageUnacceptable, CONCAT(sLeakageUnacceptable, 'R4 '));
			IF sLeakageUnacceptable = '' THEN
				R_S.vacuum_holding										:= TRUE;											// 18.a.i
				R_S.co2_sensors_off										:= TRUE;											// 19
				IF sLeakageAcceptable <> '' THEN
					sError												:= CONCAT(sLeakageAcceptable, gsVacuumPressureAcceptableBotNotIdealError);		// 18.b.i
					sMessage											:= gsReactorSetWillContinue;
				END_IF																										// else 18.a
				i6Step													:= 99;
			ELSE
				R_S.vacuum_holding										:= FALSE;											// 18.c.ii
				sReactorError											:= CONCAT(sLeakageUnacceptable, gsVacuumPressureUnacceptableError);				// 18.c.i
				sMessage												:= gsReactorSetWillPause;
			END_IF
		END_IF			
		
	80:																														// Stop process
		Cycle_Stage														:= 'evacuation.stopping';
		R_S.co2_sensors_off												:= TRUE;
		R_S.dead_air_valve												:= FALSE;
		U.dead_air_vacuum_pump											:= FALSE;
		U.product_vacuum_backfeed_valve									:= _CLOSED;
		rTime1															:= _STOPPING_TIME;
		i6Step															:= i6Step + 1;
		
	81:
		bTimer1															:= TRUE;
		IF tonTimer1.Q THEN
			bTimer1														:= FALSE;
			i6Step														:= 99;
		END_IF

	90:																														// Automatic process stopping
		Cycle_Stage														:= 'evacuation.stopping';
		R_S.co2_sensors_off												:= TRUE;
		R_S.dead_air_valve												:= FALSE;
		U.dead_air_vacuum_pump											:= FALSE;
		U.product_vacuum_backfeed_valve									:= _CLOSED;
		rTime1															:= _STOPPING_TIME;
		i6Step															:= i6Step + 1;
		
	91:
		bTimer1															:= TRUE;
		IF tonTimer1.Q THEN
			bTimer1														:= FALSE;
			i6Step														:= 99;
		END_IF
		
	98:																														// Utility error hold - cleared by P_M01
		i6Step															:= 98;
		
	99:
		IF bStopAfterEvacuation THEN
			bStop														:= TRUE;
			Stop_M01_RS													:= TRUE;											// Stop Reactor in P_M01.A_AutoMode
			bStopAfterEvacuation										:= FALSE;
		END_IF
		bEvacuationDone													:= TRUE;
		U.drainage_on													:= FALSE;
		Current_Step													:= 0;
		i6Step															:= 0;
	
END_CASE

IF i6Step > 0 AND i6Step < 80 THEN
	IF bMultiProcess THEN
		IF U.safe_shutdown_error_1 <> '' AND giSafeShutdown1RS = 0 THEN
			sSafeShutdownError1											:= U.safe_shutdown_error_1;
			giSafeShutdown1RS											:= RS_Number;
		ELSIF U.safe_shutdown_error_2 <> '' AND giSafeShutdown23RS = 0 THEN
			sSafeShutdownError2											:= U.safe_shutdown_error_2;
			giSafeShutdown23RS											:= RS_Number;
		ELSIF bEvacuationRSError AND giEvacuationErrorRS = 0 THEN															// Error occured in this reactor set
			bEvacuationRSError											:= FALSE;
			giEvacuationErrorRS											:= RS_Number;										// Save reactor set number to handle error in other reactor sets
		ELSIF giDesorptionErrorRS > 0 THEN
			bStopAfterEvacuation										:= TRUE;
		ELSIF U.os_air_unsafe_temp OR (giEvacuationErrorRS + giSafeShutdown1RS + giSafeShutdown23RS) > 0 THEN 
			Stop_Reactor_Set											:= TRUE;
		END_IF
	END_IF
	iStep																:= i6Step;
	Current_Step														:= iStep;
	A_Check_Process();
	i6Step																:= iStep;
END_IF
END_ACTION

ACTION A6_Evacuation_Test_Auto:
// Phase 0 - FB_State_Machine.A6_Evacuation_Test
// Rev 1.0 - June 3, 2024

CASE i6Step OF
	
	0:	;
	
	1:
		Cycle_Stage														:= 'evacuation.initialize';							// 1.a
		iRestartStep													:= 1;
		rTime2															:= m01.SP_evacuation_duration;
		IF U.utility_error <> '' THEN																						// 2
			sUtilityError												:= U.utility_error;
			sMessage													:= gsSystemCannotRun;
		ELSE
			rTime1														:= 10 * _seconds;
			Evac_Service_Req := TRUE;
			IF Evac_Service_Assigned THEN 
				i6Step														:= i6Step + 1;
			END_IF
		END_IF
		
	2:
		bTimer1															:= TRUE;
		//IF R_S.all_doors_closed THEN
		IF sita_bits[1].1 THEN																						// 1.c.ii
			bTimer1														:= FALSE;
			i6Step														:= 90;
		ELSIF tonTimer1.Q  AND sita_bits[1].2 THEN
			bTimer1														:= FALSE;
			sReactorError												:= gsDoorsNotClosedError;
			sMessage													:= gsReactorSetCannotRun;
		END_IF
		
	80:																														// Stop process
		Cycle_Stage														:= 'evacuation.stopping';
		rTime1															:= _STOPPING_TIME;
		i6Step															:= i6Step + 1;
		
	81:
		bTimer1															:= TRUE;
		IF tonTimer1.Q THEN
			bTimer1														:= FALSE;
			i6Step														:= 99;
		END_IF

	90:																														// Automatic process stopping
		Cycle_Stage														:= 'evacuation.stopping';
		rTime1															:= _STOPPING_TIME;
		i6Step															:= i6Step + 1;
		
	91:
		bTimer1															:= TRUE;
		IF tonTimer1.Q THEN
			bTimer1														:= FALSE;
			i6Step														:= 99;
		END_IF
		
	98:																														// Utility error hold - cleared by P_M01
		i6Step															:= 98;
		
	99:
		bEvacuationDone													:= TRUE;
		Evac_Service_Req 												:= FALSE;
		Current_Step													:= 0;
		i6Step															:= 0;
	
END_CASE

IF i6Step > 0 AND i6Step < 80 THEN
	IF bMultiProcess THEN
		IF U.safe_shutdown_error_1 <> '' AND giSafeShutdown1RS = 0 THEN
			sSafeShutdownError1											:= U.safe_shutdown_error_1;
			giSafeShutdown1RS											:= RS_Number;
		ELSIF U.safe_shutdown_error_2 <> '' AND giSafeShutdown23RS = 0 THEN
			sSafeShutdownError2											:= U.safe_shutdown_error_2;
			giSafeShutdown23RS											:= RS_Number;
		ELSIF bEvacuationRSError AND giEvacuationErrorRS = 0 THEN															// Error occured in this reactor set
			bEvacuationRSError											:= FALSE;
			giEvacuationErrorRS											:= RS_Number;										// Save reactor set number to handle error in other reactor sets
		ELSIF giDesorptionErrorRS > 0 THEN
			bStopAfterEvacuation										:= TRUE;
		ELSIF U.os_air_unsafe_temp OR (giEvacuationErrorRS + giSafeShutdown1RS + giSafeShutdown23RS) > 0 THEN 
			Stop_Reactor_Set											:= TRUE;
		END_IF
	END_IF
	iStep																:= i6Step;
	Current_Step														:= iStep;
	A_Check_Process();
	i6Step																:= iStep;
END_IF
END_ACTION

ACTION A7_Desorption:
// Phase 0 - FB_Reactor_Set.A7_Desorption
// Rev 1.0 - May 13, 2024

CASE i7Step OF
	
	0:	;
		
	1:
		Cycle_Stage														:= 'desorption.initialize';							// 4.a
		bDesorptionErrorCheck											:= FALSE;
		bSPAdjust														:= FALSE;
		iRestartStep													:= 1;
		iCycleCount														:= iCycleCount + 1;
		rTime1															:= 5 * _SECONDS;
		rTime2															:= m01.SP_steam_pressurization_and_purge_duration * _MINUTES;
		rTime3															:= rTime2 + (m01.SP_vacuum_cooling_duration * _MINUTES);
		IF R_S.reactor_pressure_error <> '' THEN
			sReactorError												:= R_S.reactor_pressure_error;
			sMessage													:= gsProcessCannotRun;
		ELSE
			i7Step														:= i7Step + 1;
		END_IF
			
	2:
		IF NOT bMultiProcess THEN
			IF NOT R_S.all_clamps_extended THEN																				// 2.a
				sReactorError											:= gsDoorClampsExtendedError;
				sMessage												:= gsProcessCannotRun;
			END_IF
		ELSE
			i7Step														:= i7Step + 1;
		END_IF

	3:
		bTimer2															:= TRUE;											// 4 - Desorption and Purge Timer
		bTimer3															:= TRUE;											// 5 - Desorption Purge and Evaporative Cooling Timer
		R_S.close_all_valves											:= TRUE;											// 6.a
		rTime1															:= _VALVE_TIME;
		i7Step															:= i7Step + 1;
		
	4:
		bTimer1															:= TRUE;
		IF R_S.valves_clear THEN
			bTimer1														:= FALSE;
			U.product_vacuum_backfeed_valve								:= _OPEN;											// 6.b
			rTime1														:= _VALVE_TIME;
			i7Step														:= i7Step + 1;
		ELSIF tonTimer1.Q THEN
			bTimer1														:= FALSE;
			sReactorError												:= SEL(R_S.steam_control_valve_closed, gsSteamControlValveError, '');
			sReactorError												:= SEL(R_S.dead_air_valve_clear, gsDeadAirValveError, sReactorError);
			sReactorError												:= SEL(R_S.purge_valve_clear, gsPurgeValveError, sReactorError); 
			sReactorError												:= SEL(R_S.cooling_valve_clear, gsCoolingValveError, sReactorError);
			sReactorError												:= SEL(R_S.steam_header_valve_clear, gsSteamHeaderValveError, sReactorError);
			sMessage													:= gsReactorSetCannotRun;
		END_IF

	5:
		bTimer1															:= TRUE;
		IF U.product_vacuum_backfeed_valve_open THEN																		// 6.a
			bTimer1														:= FALSE;
			i7Step														:= i7Step + 1;
		ELSIF tonTimer1.Q THEN
			bTimer1														:= FALSE;
			sUtilityError												:= gsProductVacuumBackfeedValveError;
			sMessage													:= gsReactorSetCannotRun;
		END_IF
	
	6:
		iStatus															:= F_LowMidHigh(m01.steam_temp_near_rs1, m01.SP_module_steam_line_low_temperature, m01.SP_module_steam_line_high_temperature, 0);
		IF NOT U.boiler_ready OR iStatus = eLow THEN																		// 7 & 8.a
			sReactorError												:= gsBoilerError;									// Stop this reactor set (no Safe Shutdown needed)
			bDesorptionRSError											:= TRUE;
		ELSIF iStatus = eHigh THEN																							// 8.c
			sSafeShutdownError2											:= gsDesorptionHighSteamLineTemp;
		ELSE																												// 8.b
			i7Step														:= i7Step + 1;
		END_IF
		
	7:
		iStatus															:= F_LowMidHigh(m01.steam_manifold_line_pres, m01.SP_module_steam_line_low_pressure, m01.SP_module_steam_line_high_pressure, 0);
		IF iStatus = eLow THEN																								// 9.a
			sReactorError												:= gsSteamPressureLowError;							// Stop this reactor set (no Safe Shutdown needed)
			bDesorptionRSError											:= TRUE;
		ELSIF iStatus = eHigh THEN																							// 9.c
			sSafeShutdownError2											:= gsSteamPressureHighError;
		ELSE																												// 9.b
			U.drainage_on												:= TRUE;											// 10
			U.product_vacuum_pump_vfd									:= u01.SP_product_vacuum_idle_vfd_percent;			// 11
			i7Step														:= i7Step + 1;
		END_IF
		
	8:	IF R_S.reactor_vacuum_status = eMid THEN																			// 12.b
			sError														:= gsReactorPressureAboveDesiredLevelError;
			sMessage													:= gsProcessWillContinue;
		ELSIF R_S.reactor_vacuum_status = eHigh THEN																		// 12.c
			sReactorError												:= gsReactorPressureAboveAcceptableLevelError;
			sMessage													:= gsReactorSetWillStop;
		ELSE																												// 12.a
			R_S.co2_outside_sensors_on									:= TRUE;											// 13
			i7Step														:= 20;
		END_IF

	20:																														//// 3.4.3.2 - Steam Pressurization
		R_S.steam_header_valve											:= TRUE;											// 1
		rTime1															:= _VALVE_TIME;
		i7Step															:= i7Step + 1;
		
	21:
		bTimer1															:= TRUE;
		IF R_S.steam_header_valve_clear THEN
			bTimer1														:= FALSE;											// 2
			rIncrementalMove											:= m01.SP_initial_maximum_steam_valve_percent_open / (m01.SP_steam_pressure_control_valve_initial_opening_duration * 120);
			rPosition													:= rIncrementalMove;
			R_S.steam_control_valve_mode								:= eManual;
			R_S.steam_control_valve										:= rPosition;
			rTime1														:= _SECONDS * 0.5;									// Half second interval update
			Cycle_Stage													:= 'desorption.pressurization.steam';				// 2.a
			i7Step														:= i7Step + 1;
		ELSIF tonTimer1.Q THEN
			bTimer1														:= FALSE;
			sSafeShutdownError2											:= gsSteamHeaderValveError;
		END_IF
		
	22:
		bTimer1															:= TRUE;
		IF tonTimer1.Q THEN
			tonTimer1(IN:= FALSE);
			rPosition													:= rPosition + rIncrementalMove;
			R_S.steam_control_valve										:= rPosition;
			IF rPosition >= m01.SP_initial_maximum_steam_valve_percent_open THEN
				 R_S.steam_control_valve								:= m01.SP_initial_maximum_steam_valve_percent_open;
				 bTimer1												:= FALSE;
				 i7Step													:= i7Step + 1;
			END_IF
		END_IF
	
	23:
		R_S.steam_control_valve_setpoint								:= m01.SP_steam_purge_pressure;						// 3
		R_S.steam_control_valve_control_point							:= R_S.average_reactor_pressure;
		R_S.steam_control_valve_mode									:= eAuto;
		i7Step															:= i7Step + 1;

	24:
		IF R_S.average_reactor_pressure >= m01.SP_start_steam_purge_reactor_pressure THEN
			i7Step														:= SEL(m01.SP_vacuum_assisted_purge, 40, 30);		// 4.a
		ELSIF tonTimer2.Q THEN																								// 4.b
			bTimer2														:= FALSE;
			sError														:= gsSteamFailedToPressurizeReactorError;
			sMessage													:= gsReactorSetWillStopAtEndOfCycle;
			Cancel_Reactor_Set											:= TRUE;
			i7Step														:= 50;
		END_IF								

		
	25:																														// 2.b
		R_S.steam_header_valve											:= FALSE;
		R_S.steam_control_valve_mode									:= eManual;
		R_S.steam_control_valve											:= 0;
		u.product_condenser												:= TRUE;
		iMaxSorbentTempErrorCount										:= iMaxSorbentTempErrorCount + 1;
		sError															:= gsSorbentTemperatureError;
		sMessage														:= gsReactorSetWillContinue;
		IF iMaxSorbentTempErrorCount / iCycleCount >= 0.15 THEN
			sMessage													:= gsReactorSetWillStopAtEndOfCycle;
			Cancel_Reactor_Set											:= TRUE;
		END_IF
		i7Step															:= i7Step + 1;
		
	26:
		IF tonTimer2.Q THEN
			bTimer2														:= FALSE;
			i7Step														:= 50;
		END_IF

	
	27:																														// 2.c
		R_S.steam_header_valve											:= FALSE;
		R_S.steam_control_valve_mode									:= eManual;
		R_S.steam_control_valve											:= 0;
		R_S.steam_control_valve_mode									:= eManual;
		R_S.steam_control_valve											:= 0;
		sSafeShutdownError2												:= gsSteamPressureHighError;

		
	28:																														// 2.d
		u.product_vacuum_pump_isolation_valve							:= FALSE;
		R_S.purge_valve													:= FALSE;
		R_S.cooling_valve												:= FALSE;
		R_S.steam_header_valve											:= FALSE;
		u.product_vacuum_pump_vfd										:= u01.SP_product_vacuum_idle_vfd_percent;
		sSafeShutdownError2												:= gsPostCondenserLineHighTempError;
	

//// 3.4.3.3 - Vacuum Assisted Purge
	30:																													
		u.product_vacuum_bypass_valve									:= FALSE;											// 1.a
		rTime1															:= _VALVE_TIME;
		i7Step															:= i7Step + 1;
		
	31:
		bTimer1															:= TRUE;
		IF u.product_vacuum_bypass_valve_clear THEN
			bTimer1														:= FALSE;
			u.product_vacuum_pump_vfd									:= u01.SP_product_vacuum_running_vfd_percent;		// 1.b
			u.product_condenser											:= TRUE;
			u.product_vacuum_pump_isolation_valve						:= TRUE;
			u.product_vacuum_outlet_isolation_valve						:= TRUE;
			u.product_blower											:= TRUE;
			u.purge_product_pre_condenser_valve							:= TRUE;
			i7Step														:= i7Step + 1;
		ELSIF tonTimer1.Q THEN
			;	///@ valve error TBD
		END_IF

	32:
		u.product_vacuum_backfeed_valve_setpoint						:= m01.SP_steam_purge_pressure;						// 2
		u.product_vacuum_backfeed_valve_mode							:= eAuto;
		rSP1															:= m01.SP_steam_purge_pressure;
		rSP1															:= rSP1 - (rSP1 * m01.SP_percent_from_steam_purge_target_pressure * 0.01);
		i7Step															:= i7Step + 1;
		
	33:
		IF u.product_vacuum_pres >= rSP1 THEN																				// 3
			R_S.purge_valve												:= TRUE;											// 3.a
			Cycle_Stage													:= 'desorption.steam_vacuum_assisted';				// 3.b
			i7Step														:= i7Step + 1;
		ELSIF R_S.sorbent_high_temp > m01.SP_maximum_target_sorbent_temperature_during_purge AND NOT bSPAdjust THEN			// 2.a
			rSP1														:= m01.SP_steam_purge_pressure - m01.SP_steam_purge_pressure_decrease;
			u.product_vacuum_backfeed_valve_setpoint					:= rSP1;
			rSP1														:= rSP1 - (rSP1 * m01.SP_percent_from_steam_purge_target_pressure * 0.01);
			bSPAdjust													:= TRUE;
		ELSIF tonTimer2.Q THEN																								// 3.c
			bTimer2														:= FALSE;
			sSafeShutdownError3											:= gsDesorptionPurgeLinePressureError;
		END_IF
		
	34:
		IF tonTimer2.Q THEN																									// 4
			R_S.steam_header_valve										:= FALSE;											// 4.a
			R_S.steam_control_valve_mode								:= eManual;											// 4.a.i
			R_S.steam_control_valve										:= 0;
			bTimer2														:= FALSE;											// 4.b
			i7Step														:= 50;						
		END_IF

		
//// 3.4.3.4 - No vacuum purge			
	40:																														
		u.product_vacuum_backfeed_valve_mode							:= eManual;											// 1.a
		u.product_vacuum_backfeed_valve									:= 0;
		u.product_condenser												:= TRUE;
		u.product_vacuum_bypass_valve									:= TRUE;
		u.purge_product_pre_condenser_valve								:= TRUE;
		u.product_blower												:= TRUE;
		i7Step															:= i7Step + 1;
	
	41:
		IF u.pre_condenser_line_pres < R_S.average_reactor_pressure THEN													// 2
			R_S.purge_valve												:= TRUE;											// 2.b
			Cycle_Stage													:= 'desorption.steam_no_vacuum';					// 2.c
			i7Step														:= i7Step + 1;
		ELSIF tonTimer2.Q THEN
			bTimer2														:= FALSE;
			sSafeShutdownError2											:= gsDesorptionPurgeLinePressureError;
		END_IF
	
	42:
		R_S.steam_control_valve_setpoint								:= m01.SP_steam_purge_pressure;						// 3
		R_S.steam_control_valve_control_point							:= u.product_vacuum_pres;		///@ u.pre_condenser_line_pres????
		R_S.steam_control_valve_mode									:= eAuto;
		i7Step															:= i7Step + 1;
		
	43:
		IF tonTimer2.Q THEN																									// 4
			R_S.steam_header_valve										:= FALSE;											// 4.a
			R_S.steam_control_valve_mode								:= eManual;											// 4.a.i
			R_S.steam_control_valve										:= 0;
			bTimer2														:= FALSE;											// 4.b
			i7Step														:= 99;						
		END_IF


//// 3.4.3.5 - Vacuum cooling	
	50:
		R_S.purge_valve													:= FALSE;											// 1.a
		u.purge_product_pre_condenser_valve								:= FALSE;
		u.product_vacuum_bypass_valve									:= FALSE;
		u.product_vacuum_pump_isolation_valve							:= TRUE;
		u.product_vacuum_backfeed_valve									:= _CLOSED;
		u.product_vacuum_backfeed_valve_mode							:= eManual;
		u.product_vacuum_outlet_isolation_valve							:= TRUE;
		u.product_vacuum_pump_vfd										:= u01.SP_product_vacuum_running_vfd_percent;
		u.cooling_line_pre_condenser_valve								:= TRUE;
		rTime1															:= _VALVE_TIME;
		i7Step															:= i7Step + 1;
		
	51:
		bTimer1															:= TRUE;
		bPass1															:= R_S.purge_valve_clear;
		bPass1															:= u.purge_product_pre_condenser_valve_clear;
		bPass3															:= u.product_vacuum_bypass_valve_clear;
		bPass4															:= u.product_vacuum_backfeed_valve_closed;
		bPass5															:= u.product_vacuum_outlet_isolation_valve_clear;
		bPass6															:= u.cooling_line_pre_condenser_valve_clear;
		IF bPass1 AND bPass2 AND bPass3 AND bPass4 AND bPass5 AND bPass6 THEN 
			bTimer1														:= FALSE;
			i7Step														:= i7Step + 1;
		ELSIF tonTimer1.Q THEN
			;	///@ Valve error
		END_IF

	52:
		IF u.product_vacuum_pres < R_S.average_reactor_pressure THEN														///@ Timer function?
			R_S.cooling_valve											:= TRUE;											// 1.b
			Cycle_Stage													:= 'desorption.cooling';							// 1.c
			i7Step														:= i7Step + 1;			
		END_IF

	53:
		IF tonTimer3.Q THEN																									// 2
			u.product_blower											:= FALSE;											// 3
			u.product_vacuum_pump_isolation_valve						:= FALSE;											// 4.a
			u.cooling_line_pre_condenser_valve							:= FALSE;
			R_S.cooling_valve											:= FALSE;
			u.product_vacuum_pump_vfd									:= u01.SP_product_vacuum_idle_vfd_percent;			// 5
			u.product_vacuum_backfeed_valve								:= _OPEN;											// 5.a
			Cycle_Stage													:= 'desorption.wrap_up';							// 5.b
			i7Step														:= i7Step + 1;
		END_IF
			
	54:
		iStatus															:= F_LowMidHigh(R_S.average_reactor_pressure, m01.SP_vacuum_cooling_target_pressure, m01.SP_vacuum_cooling_unacceptable_pressure, 0);	// 6
		IF iStatus = eHigh THEN																								// 6.c
			sSafeShutdownError3											:= gsVacuumPressureUnacceptableError;
		ELSIF iStatus = eMid THEN																							// 6.b
			sError														:= gsVacuumCoolingAcceptableButNotIdealError;
			sMessage													:= gsProcessWillContinue;
		END_IF
		i7Step															:= i7Step + 1;										// 6.a
		
	55:
		R_S.retract_all_clamps											:= TRUE;
		rTime1															:= m01.SP_clampsretract_timedelay * _MINUTES;
		i7Step															:= i7Step + 1;
		
	56:
		IF R_S.all_clamps_retracted THEN
			bTimer1														:= FALSE;
			bTimer2														:= FALSE;
			bTimer3														:= FALSE;
			R_S.co2_sensors_off											:= TRUE;
			i7Step														:= 99;
		ELSIF tonTimer1.Q THEN
			sPauseError													:= gsClampRetractError;
			sMessage													:= gsReactorSetWillStop;
		END_IF
		
		
	80:																														// Manual process closing
		Cycle_Stage														:= 'desorption.stopping';
		U.product_vacuum_backfeed_valve									:= _CLOSED;
		rTime1															:= _STOPPING_TIME;
		i7Step															:= 81;
		
	81:
		bTimer1															:= TRUE;
		IF tonTimer1.Q THEN
			bTimer1														:= FALSE;
			i7Step														:= 99;
		END_IF

	90:																														// Automatic process stopping
		Cycle_Stage														:= 'desorption.stopping';
		U.product_vacuum_backfeed_valve									:= _CLOSED;											///@ Close valves & turn off pumps
		rTime1															:= _STOPPING_TIME;
		i7Step															:= 91;
		
	91:
		bTimer1															:= TRUE;
		IF tonTimer1.Q THEN
			bTimer1														:= FALSE;
			i7Step														:= 99;
		END_IF
		
	98:																														// Utility error hold - cleared by P_M01
		i7Step															:= 98;
		
	99:
		IF bStopAfterDesorption THEN
			bStop														:= TRUE;
			Stop_M01_RS													:= TRUE;											// Stop Reactor in P_M01.A_AutoMode
			bStopAfterDesorption										:= FALSE;
		END_IF
		bDesorptionDone													:= TRUE;
		Current_Step													:= 0;
		i7Step															:= 0;
	
END_CASE

IF i7Step > 0 AND i7Step < 80 THEN
	IF bMultiProcess THEN
		IF U.safe_shutdown_error_1 <> '' AND giSafeShutdown1RS = 0 THEN
			sSafeShutdownError1											:= U.safe_shutdown_error_1;
			giSafeShutdown1RS											:= RS_Number;
		ELSIF U.safe_shutdown_error_2 <> '' AND giSafeShutdown23RS = 0 THEN
			sSafeShutdownError2											:= U.safe_shutdown_error_2;
			giSafeShutdown23RS											:= RS_Number;
		ELSIF bDesorptionRSError AND giDesorptionErrorRS = 0 THEN
			bDesorptionRSError											:= FALSE;
			giDesorptionErrorRS											:= RS_Number;
			sMessage													:= gsReactorSetWillStopEvacWillFinishOthersWillCompleteCycle;
		ELSIF (sSafeShutdownError2 <> '' OR sSafeShutdownError3 <> '') AND giSafeShutdown23RS = 0 THEN
			giSafeShutdown23RS											:= RS_Number;
		ELSIF (giDesorptionErrorRS + giSafeShutdown23RS) > 0 THEN
			Stop_Reactor_Set											:= TRUE;
		ELSIF (giEvacuationErrorRS + giSafeShutdown1RS) > 0 THEN
			Cancel_Reactor_Set											:= TRUE;
		ELSIF U.os_air_unsafe_temp THEN																							// 5.e
			bStopAfterDesorption										:= TRUE;
		END_IF
		IF NOT bDesorptionErrorCheck THEN
			IF R_S.steam_header_valve_not_closed THEN
				IF R_S.desorption_high_temp_count > _DESORP_MAX_COUNT THEN														//3.4.3.2_2.b
					bDesorptionErrorCheck								:= TRUE;
					i7Step												:= 25;
				ELSIF R_S.average_reactor_pressure > m01.SP_maximum_safe_reactor_steam_pressure THEN							//3.4.3.2_2.c
					bDesorptionErrorCheck								:= TRUE;
					i7Step												:= 27;
				END_IF
			ELSIF NOT u.product_vacuum_pump_isolation_valve_closed THEN
				IF u.post_condenser_line_temp > u01.SP_maximum_inlet_product_vacuum_temperature THEN							//3.4.3.2_2.d
					bDesorptionErrorCheck								:= TRUE;
					i7Step												:= 28;
				END_IF
			END_IF
		END_IF
	END_IF
	iStep																:= i7Step;
	Current_Step														:= iStep;
	A_Check_Process();
	i7Step																:= iStep;
END_IF
END_ACTION

ACTION A7_Desorption_Test:
// Phase 0 - FB_Reactor_Set.A7_Desorption_Test
// Rev 1.0 - June 3, 2024

CASE i7Step OF
	
	0:	;
		
	1:
		Cycle_Stage														:= 'desorption.initialize';							// 4.a
		rTime1															:= 5 * _SECONDS;
		rTime2															:= m01.SP_steam_pressurization_and_purge_duration * _MINUTES;
		rTime3															:= rTime2 + (m01.SP_vacuum_cooling_duration * _MINUTES);
		IF R_S.reactor_pressure_error <> '' THEN
			sReactorError												:= R_S.reactor_pressure_error;
			sMessage													:= gsProcessCannotRun;
		ELSE
			i7Step														:= i7Step + 1;
		END_IF
			
	2:
		bTimer1															:= TRUE;
		U.cooling_line_pre_condenser_valve								:= TRUE;
		U.purge_product_pre_condenser_valve								:= TRUE;
		U.product_vacuum_pump_isolation_valve 							:= TRUE;
		U.product_vacuum_outlet_isolation_valve 						:= TRUE;
		U.product_vacuum_backfeed_valve									:= 50;											// 6.b
		rTime1															:= _VALVE_TIME;
		i7Step															:= i7Step + 1;

	3:
		//bTimer1															:= TRUE;
		IF U.purge_product_line_pres < m01.SP_start_steam_purge_reactor_pressure AND U.pre_condenser_line_pres < m01.SP_start_steam_purge_reactor_pressure THEN
			U.steam_header_volume_total_enable							:= TRUE;
			U.cooling_line_pre_condenser_valve							:= FALSE;
			R_S.steam_header_valve										:= TRUE;
			R_S.steam_control_valve										:= _OPEN;
			i7Step														:= i7Step + 1;
		END_IF
		
	4:
		IF R_S.average_reactor_pressure >= m01.SP_maximum_target_steam_pressure THEN
			R_S.purge_valve 											:= TRUE;
			U.product_vacuum_pump_vfd									:= u01.SP_product_vacuum_running_vfd_percent;
			U.product_vacuum_backfeed_valve								:= u01.SP_product_vacuum_backfeed_valve;
			i7Step														:= i7Step + 1;
		END_IF
		
	5:
		bTimer2															:= TRUE;
		IF (U01.SP_mass_flow_totalizer <> 0 AND U01.SP_mass_flow_totalizer >= u01.steam_header_volume_total) OR tonTimer2.Q THEN
			bTimer2														:= FALSE;
			i7Step														:= i7Step + 1;
		END_IF
	
	6:
		R_S.steam_header_valve											:= FALSE;
		R_S.purge_valve													:= FALSE;
		R_S.steam_control_valve											:= _CLOSED;
		U.product_vacuum_backfeed_valve									:= _CLOSED;
		U.cooling_line_pre_condenser_valve								:= FALSE;
		U.purge_product_pre_condenser_valve								:= FALSE;
		U.product_vacuum_pump_vfd										:= 100;
		U.product_blower_vfd											:= 100;
		R_S.cooling_valve												:= TRUE;
		i7Step															:= i7Step + 1;
		
	7:
		IF R_S.sorbent_high_temp <= 58 THEN
			R_S.cooling_valve											:= FALSE;
			U.product_vacuum_backfeed_valve								:= 50;
			U.product_vacuum_pump_vfd									:= 50;
			u.product_blower_vfd										:= 0;
			i7Step														:= 99;
		END_IF
		
	80:																														// Manual process closing
		Cycle_Stage														:= 'desorption.stopping';
		U.product_vacuum_backfeed_valve									:= _CLOSED;
		rTime1															:= _STOPPING_TIME;
		i7Step															:= 81;
		
	81:
		bTimer1															:= TRUE;
		IF tonTimer1.Q THEN
			bTimer1														:= FALSE;
			i7Step														:= 99;
		END_IF

	90:																														// Automatic process stopping
		Cycle_Stage														:= 'desorption.stopping';
		U.product_vacuum_backfeed_valve									:= _CLOSED;											///@ Close valves & turn off pumps
		rTime1															:= _STOPPING_TIME;
		i7Step															:= 91;
		
	91:
		bTimer1															:= TRUE;
		IF tonTimer1.Q THEN
			bTimer1														:= FALSE;
			i7Step														:= 99;
		END_IF
		
	98:																														// Utility error hold - cleared by P_M01
		i7Step															:= 98;
		
	99:
		IF bStopAfterDesorption THEN
			bStop														:= TRUE;
			Stop_M01_RS													:= TRUE;											// Stop Reactor in P_M01.A_AutoMode
			bStopAfterDesorption										:= FALSE;
		END_IF
		bDesorptionDone													:= TRUE;
		U.steam_header_volume_total_enable								:= FALSE;
		Current_Step													:= 0;
		i7Step															:= 0;
	
END_CASE

IF i7Step > 0 AND i7Step < 80 THEN
	IF bMultiProcess THEN
		IF U.safe_shutdown_error_1 <> '' AND giSafeShutdown1RS = 0 THEN
			sSafeShutdownError1											:= U.safe_shutdown_error_1;
			giSafeShutdown1RS											:= RS_Number;
		ELSIF U.safe_shutdown_error_2 <> '' AND giSafeShutdown23RS = 0 THEN
			sSafeShutdownError2											:= U.safe_shutdown_error_2;
			giSafeShutdown23RS											:= RS_Number;
		ELSIF bDesorptionRSError AND giDesorptionErrorRS = 0 THEN
			bDesorptionRSError											:= FALSE;
			giDesorptionErrorRS											:= RS_Number;
			sMessage													:= gsReactorSetWillStopEvacWillFinishOthersWillCompleteCycle;
		ELSIF (sSafeShutdownError2 <> '' OR sSafeShutdownError3 <> '') AND giSafeShutdown23RS = 0 THEN
			giSafeShutdown23RS											:= RS_Number;
		ELSIF (giDesorptionErrorRS + giSafeShutdown23RS) > 0 THEN
			Stop_Reactor_Set											:= TRUE;
		ELSIF (giEvacuationErrorRS + giSafeShutdown1RS) > 0 THEN
			Cancel_Reactor_Set											:= TRUE;
		ELSIF U.os_air_unsafe_temp THEN																							// 5.e
			bStopAfterDesorption										:= TRUE;
		END_IF
		IF NOT bDesorptionErrorCheck THEN
			IF R_S.steam_header_valve_not_closed THEN
				IF R_S.desorption_high_temp_count > _DESORP_MAX_COUNT THEN														//3.4.3.2_2.b
					bDesorptionErrorCheck								:= TRUE;
					i7Step												:= 25;
				ELSIF R_S.average_reactor_pressure > m01.SP_maximum_safe_reactor_steam_pressure THEN							//3.4.3.2_2.c
					bDesorptionErrorCheck								:= TRUE;
					i7Step												:= 27;
				END_IF
			ELSIF NOT u.product_vacuum_pump_isolation_valve_closed THEN
				IF u.post_condenser_line_temp > u01.SP_maximum_inlet_product_vacuum_temperature THEN							//3.4.3.2_2.d
					bDesorptionErrorCheck								:= TRUE;
					i7Step												:= 28;
				END_IF
			END_IF
		END_IF
	END_IF
	iStep																:= i7Step;
	Current_Step														:= iStep;
	A_Check_Process();
	i7Step																:= iStep;
END_IF
END_ACTION

ACTION A7_Desorption_Test_Auto:
// Phase 0 - FB_Reactor_Set.A7_Desorption_Test
// Rev 1.0 - June 3, 2024

CASE i7Step OF
	
	0:	;
		
	1:
		Cycle_Stage														:= 'desorption.initialize';							// 4.a
		rTime1															:= 5 * _SECONDS;
		rTime2															:= m01.SP_steam_pressurization_and_purge_duration * _MINUTES;
		rTime3															:= rTime2 + (m01.SP_vacuum_cooling_duration * _MINUTES);
		Steam_Service_Req												:= TRUE;
		IF Steam_Service_Assigned THEN 
			i7Step															:= i7Step + 1;
		END_IF
		
			
	2:
		bTimer1															:= TRUE;
		IF sita_bits[2].1 THEN 
			bTimer1														:= FALSE;
			i7Step														:= 90;
		ELSIF tonTimer1.Q AND  sita_bits[2].2 THEN 
			bTimer1														:= FALSE;
			sReactorError												:= 'Desorption Error';
			sMessage													:= 'Auto Test';
		END_IF

	
		
	80:																														// Manual process closing
		Cycle_Stage														:= 'desorption.stopping';
		U.product_vacuum_backfeed_valve									:= _CLOSED;
		rTime1															:= _STOPPING_TIME;
		i7Step															:= 81;
		
	81:
		bTimer1															:= TRUE;
		IF tonTimer1.Q THEN
			bTimer1														:= FALSE;
			i7Step														:= 99;
		END_IF

	90:																														// Automatic process stopping
		Cycle_Stage														:= 'desorption.stopping';
		rTime1															:= _STOPPING_TIME;
		i7Step															:= 91;
		
	91:
		bTimer1															:= TRUE;
		IF tonTimer1.Q THEN
			bTimer1														:= FALSE;
			i7Step														:= 99;
		END_IF
		
	98:																														// Utility error hold - cleared by P_M01
		i7Step															:= 98;
		
	99:
		IF bStopAfterDesorption THEN
			bStop														:= TRUE;
			Stop_M01_RS													:= TRUE;											// Stop Reactor in P_M01.A_AutoMode
			bStopAfterDesorption										:= FALSE;
		END_IF
		bDesorptionDone													:= TRUE;
		IF NOT bMultiProcess THEN
			Steam_Service_Req											:= FALSE;
		END_IF
		Current_Step													:= 0;
		i7Step															:= 0;
	
END_CASE

IF i7Step > 0 AND i7Step < 80 THEN
	IF bMultiProcess THEN
		IF U.safe_shutdown_error_1 <> '' AND giSafeShutdown1RS = 0 THEN
			sSafeShutdownError1											:= U.safe_shutdown_error_1;
			giSafeShutdown1RS											:= RS_Number;
		ELSIF U.safe_shutdown_error_2 <> '' AND giSafeShutdown23RS = 0 THEN
			sSafeShutdownError2											:= U.safe_shutdown_error_2;
			giSafeShutdown23RS											:= RS_Number;
		ELSIF bDesorptionRSError AND giDesorptionErrorRS = 0 THEN
			bDesorptionRSError											:= FALSE;
			giDesorptionErrorRS											:= RS_Number;
			sMessage													:= gsReactorSetWillStopEvacWillFinishOthersWillCompleteCycle;
		ELSIF (sSafeShutdownError2 <> '' OR sSafeShutdownError3 <> '') AND giSafeShutdown23RS = 0 THEN
			giSafeShutdown23RS											:= RS_Number;
		ELSIF (giDesorptionErrorRS + giSafeShutdown23RS) > 0 THEN
			Stop_Reactor_Set											:= TRUE;
		ELSIF (giEvacuationErrorRS + giSafeShutdown1RS) > 0 THEN
			Cancel_Reactor_Set											:= TRUE;
		ELSIF U.os_air_unsafe_temp THEN																							// 5.e
			bStopAfterDesorption										:= TRUE;
		END_IF
		IF NOT bDesorptionErrorCheck THEN
			IF R_S.steam_header_valve_not_closed THEN
				IF R_S.desorption_high_temp_count > _DESORP_MAX_COUNT THEN														//3.4.3.2_2.b
					bDesorptionErrorCheck								:= TRUE;
					i7Step												:= 25;
				ELSIF R_S.average_reactor_pressure > m01.SP_maximum_safe_reactor_steam_pressure THEN							//3.4.3.2_2.c
					bDesorptionErrorCheck								:= TRUE;
					i7Step												:= 27;
				END_IF
			ELSIF NOT u.product_vacuum_pump_isolation_valve_closed THEN
				IF u.post_condenser_line_temp > u01.SP_maximum_inlet_product_vacuum_temperature THEN							//3.4.3.2_2.d
					bDesorptionErrorCheck								:= TRUE;
					i7Step												:= 28;
				END_IF
			END_IF
		END_IF
	END_IF
	iStep																:= i7Step;
	Current_Step														:= iStep;
	A_Check_Process();
	i7Step																:= iStep;
END_IF
END_ACTION

END_FUNCTION_BLOCK

// ---- POUs/Functions/F_SetProcess.TcPOU
FUNCTION F_SetProcess : INT
VAR_INPUT
	Process																: INT;
	Mode																: STRING;
END_VAR
VAR
END_VAR

// F_SetProcess
// Rev 1.0 - May 3, 2024

F_SetProcess															:= FIND(INT_TO_STRING(Process), Mode);

END_FUNCTION

// ---- POUs/P_Alarms.TcPOU
PROGRAM P_Alarms
VAR
	i																	: INT;
	sitaBits : DWORD;
	sitaAlarm : STRING;
	sitaMsg : STRING;
	sitaTmr : STRING;
	sitaRTrig : R_TRIG;
	alarm_number : INT;
END_VAR

// Phase 0 - P_Alarms
// Rev 1.0 - February 26, 2024
FOR i := 1 TO alarm_number DO 
	IF gsAlarms[i] <> '' THEN 
		m01.ts_Alarm			:= gsAlarms[i];
		m01.ts_User_Message		:= gsMessages[i];
		m01.tb_Alarm_Active		:= TRUE;
		EXIT ;
	END_IF
END_FOR


IF m01.tb_Acknowledge_Alarm THEN
	FOR i := 1 TO alarm_number DO 
		IF gsAlarms[i] <> '' THEN                     	    	
			gsAlarms[i] 													:= '';
			gsMessages[i]													:= '';
			EXIT ;
		END_IF
	END_FOR
	m01.tb_Acknowledge_Alarm := FALSE;                                	    		
END_IF                                      	    	

IF m01.tb_Clear_Alarm_All THEN
	FOR i := 1 TO alarm_number DO                      	    	
		gsAlarms[i] 													:= '';
		gsMessages[i]													:= '';	
		m01.tb_Clear_Alarm_All											:= FALSE;		
	END_FOR                                 	    	
END_IF

giAlarmCount := M_GetAlarmsCount(); 

IF giAlarmCount = 0 THEN
	m01.ts_Alarm			:= '';
	m01.ts_User_Message		:= '';
	m01.tb_Alarm_Active		:= FALSE;
	alarm_number			:= 0;
END_IF
                                            	    	
FOR i := 1 TO _ALARM_COUNT DO 
	m01.processAlarms[i] := gsAlarms[i];
	m01.processAlarmsMessage[i] := gsMessages[i];
END_FOR

sitaRTrig(CLK := sitaBits.0);
IF sitaRTrig.Q THEN 
	M_Add_Alarm('UnitTest-',sitaAlarm,sitaMsg);
	sitaBits.0 := FALSE;
END_IF

METHOD M_Add_Alarm 			: BOOL
VAR_INPUT
	Unit																: STRING;
	Alarm																: STRING;
	Message																: STRING;
END_VAR
VAR
END_VAR
// Phase 0 - P_Alarms.M_Add_Alarm
// Rev 1.0 - January 31, 2024


IF alarm_number < _ALARM_COUNT THEN
	alarm_number													:= alarm_number + 1;
	gsMessages[alarm_number]										:= Message;
	gsAlarms[alarm_number]											:= CONCAT(Unit, Alarm);
END_IF
M_Add_Alarm															:= TRUE;
END_METHOD

METHOD M_Check_Error : BOOL
VAR_INPUT
	Error_In															: BOOL;
	Latch																: BOOL;
	Unit																: STRING;
	Alarm																: STRING;
	Message																: STRING;
END_VAR
VAR
	Error_Out															: BOOL;
END_VAR
// Phase 0 - P_Alarms.M_Check_Error
// Rev 1.0 - March 20, 2024

IF m01.tb_Auto_Mode_On THEN

	Error_Out																:= Latch;
	IF Error_In THEN
		IF NOT Error_Out THEN
			Error_Out														:= TRUE;
			P_Alarms.M_Add_Alarm(Unit, Alarm, Message);
		END_IF
	ELSE
		Error_Out															:= FALSE;
	END_IF
	M_Check_Error															:= Error_Out;

END_IF
END_METHOD

METHOD M_GetAlarmsCount : INT
VAR
	alarmCount : INT := 0 ;
END_VAR

FOR i := 0 TO alarm_number DO 
	IF gsAlarms[i] <> '' THEN 
		alarmCount := alarmCount + 1;
	END_IF
END_FOR
M_GetAlarmsCount := alarmCount;
END_METHOD

END_PROGRAM

// ---- POUs/Functions/F_Concat3.TcPOU
FUNCTION F_Concat3 : STRING
VAR_INPUT
	s1																	: STRING;
	s2																	: STRING;
	s3																	: STRING;
END_VAR
VAR
END_VAR

// F_Concat3
// Rev 1.0 - January 10, 2024

F_Concat3																:= CONCAT(s1, s2);
F_Concat3																:= CONCAT(F_Concat3, s3);

END_FUNCTION

// ---- POUs/Reactor_Set_Function_Blocks/FB_Reactor_Set_IO.TcPOU
FUNCTION_BLOCK FB_Reactor_Set_IO
VAR_IN_OUT
	condensate_pump_hmi													: BOOL;
	condensate_pump_plc													: BOOL;
	dead_air_valve_hmi													: BOOL;
	dead_air_valve_plc													: BOOL;
	purge_valve_hmi														: BOOL;
	purge_valve_plc														: BOOL;
	cooling_valve_hmi													: BOOL;
	cooling_valve_plc													: BOOL;
	steam_header_valve_hmi												: BOOL;
	steam_header_valve_plc												: BOOL;
	steam_control_valve_hmi												: REAL;
	steam_control_valve_plc												: REAL;
	steam_control_valve_mode_hmi										: INT;
	steam_control_valve_mode_plc										: INT;
END_VAR
VAR_INPUT
	power_control_in													: BOOL;
	power_control_fdbk_no												: BOOL;
	power_control_fdbk_nc												: BOOL;
	condensate_lsl_in													: BOOL;
	condensate_lsh_in													: BOOL;
	close_valves														: BOOL;
	rs_close_valves														: BOOL;
	dead_air_valve_open													: BOOL;
	dead_air_valve_closed												: BOOL;
	purge_valve_open													: BOOL;
	purge_valve_closed													: BOOL;
	cooling_valve_open													: BOOL;
	cooling_valve_closed												: BOOL;
	steam_header_valve_open												: BOOL;
	steam_header_valve_closed											: BOOL;
	reactor_over_max_pressure											: BOOL;
	PCV_01_position														: INT;
	status_in															: INT;
	steam_control_valve_setpoint										: REAL;
	steam_control_valve_control_point									: REAL;
	steam_control_valve_loop_time										: REAL;
	steam_control_valve_kp												: REAL;
	steam_control_valve_ki												: REAL;
	steam_control_valve_iband											: REAL;
	steam_control_valve_base											: INT;
	steam_control_valve_base_adjust										: INT;
	steam_control_valve_error											: BOOL;
END_VAR
VAR_OUTPUT
	power_control_out													: BOOL;
	PWR_01																: BOOL;
	condensate_lsl_out													: BOOL;
	condensate_lsh_out													: BOOL;
	P_01																: BOOL;
	condensate_pump_cmd_status											: BOOL;
	XV_04																: BOOL;
	dead_air_valve_open_cmd_status										: BOOL;
	dead_air_valve_clear												: BOOL;
	XV_05																: BOOL;
	purge_valve_open_cmd_status											: BOOL;
	purge_valve_clear													: BOOL;
	XV_06																: BOOL;
	cooling_valve_open_cmd_status										: BOOL;
	cooling_valve_clear													: BOOL;
	XV_07																: BOOL;
	steam_header_valve_open_cmd_status									: BOOL;
	steam_header_valve_clear											: BOOL;
	steam_header_valve_not_closed										: BOOL;
	PCV_01																: INT;
	steam_control_valve_current_mode									: INT;	
	steam_control_valve_position										: REAL;
	steam_control_valve_closed											: BOOL;
	valves_clear														: BOOL;
	status_out															: STRING;
	sorbent_high_temp													: REAL;
END_VAR
VAR
	fb_Condensate_Pump													: FB_Digital_Out();
	fb_Dead_Air_Valve													: FB_Digital_Out();
	fb_PurgeValve														: FB_Digital_Out();
	fb_Cooling_Valve													: FB_Digital_Out();
	fb_Steam_Header_Valve												: FB_Digital_Out();
	fb_Steam_Control_Valve_Mode											: FB_Integer_Out();
	fb_Steam_Control_Valve												: FB_Analog_Out();
	fb_Steam_Control_Valve_PI											: FB_PI_Control();
	
	bSteamHeaderValve													: BOOL;
	
END_VAR

// Phase 0 - FB_Reactor_Set_IO
// Rev 1.0 - April 30, 2024

power_control_out														:= power_control_fdbk_no AND NOT power_control_fdbk_nc AND NOT PWR_01 ;
PWR_01																	:= power_control_in;

status_out																:= SEL(status_in >= 0 AND status_in < 40, Main.sStatusLabel[40], Main.sStatusLabel[status_in]);

condensate_lsl_out														:= condensate_lsl_in;
condensate_lsh_out														:= condensate_lsh_in;

fb_Condensate_Pump(Input1:= condensate_pump_hmi, Input2:= condensate_pump_plc, Output=> P_01);
condensate_pump_cmd_status												:= P_01;

IF close_valves OR rs_close_valves THEN
	dead_air_valve_plc													:= FALSE;
	purge_valve_plc														:= FALSE;
	cooling_valve_hmi													:= FALSE;
	steam_header_valve_hmi												:= FALSE;
	close_valves														:= FALSE;
	rs_close_valves														:= FALSE;
END_IF

fb_Dead_Air_Valve(Input1:= dead_air_valve_hmi, Input2:= dead_air_valve_plc, Output=> XV_04);
dead_air_valve_open_cmd_status											:= XV_04;
dead_air_valve_clear													:= F_ValveClear(dead_air_valve_plc, dead_air_valve_open, dead_air_valve_closed);

fb_PurgeValve(Input1:= purge_valve_hmi, Input2:= purge_valve_plc, Output=> XV_05);
XV_05																	:= purge_valve_plc;
purge_valve_open_cmd_status												:= purge_valve_plc;
purge_valve_clear														:= F_ValveClear(purge_valve_plc, purge_valve_open, purge_valve_closed);

fb_Cooling_Valve(Input1:= cooling_valve_hmi, Input2:= cooling_valve_plc, Output=> XV_06);
XV_06																	:= cooling_valve_plc;
cooling_valve_open_cmd_status											:= cooling_valve_plc;
cooling_valve_clear														:= F_ValveClear(cooling_valve_plc, cooling_valve_open, cooling_valve_closed);

fb_Steam_Header_Valve(Input1:= steam_header_valve_hmi, Input2:= steam_header_valve_plc, Output=> bSteamHeaderValve);
XV_07																	:= SEL(m01.tb_Auto_Mode_On, bSteamHeaderValve AND NOT reactor_over_max_pressure, bSteamHeaderValve);
steam_header_valve_open_cmd_status										:= XV_07;
steam_header_valve_clear												:= F_ValveClear(steam_header_valve_plc, steam_header_valve_open, steam_header_valve_closed);
steam_header_valve_not_closed											:= NOT steam_header_valve_closed;

fb_Steam_Control_Valve(Input1:= steam_control_valve_hmi, Input2:= steam_control_valve_plc);
fb_Steam_Control_Valve_Mode(Input1:= steam_control_valve_mode_hmi, Input2:= steam_control_valve_mode_plc);
fb_Steam_Control_Valve_PI(	Setpoint									:= steam_control_valve_setpoint,
							Control										:= steam_control_valve_control_point,
							Error										:= steam_control_valve_error,
							Reverse										:= FALSE,
							Kp											:= steam_control_valve_kp,           
							Ki											:= steam_control_valve_ki,           
							BaseAdjust									:= steam_control_valve_base_adjust,  
							LoopTime									:= steam_control_valve_loop_time,    
							IBand										:= steam_control_valve_iband,        
							Base										:= steam_control_valve_base,         
							Mode										:= steam_control_valve_mode_plc,
							Input										:= steam_control_valve_plc,
							Mode_Out									=> steam_control_valve_current_mode, 
							Output										=> PCV_01);

steam_control_valve_position											:= INT_TO_REAL(PCV_01_position) / _PERCENT_FACTOR; 
steam_control_valve_closed												:= steam_control_valve_position <= _VALVE_CLOSED;

valves_clear															:= dead_air_valve_clear AND purge_valve_clear AND cooling_valve_clear AND steam_header_valve_clear;

END_FUNCTION_BLOCK

// ---- POUs/Reactor_Set_Function_Blocks/FB_Reactor_IO.TcPOU
FUNCTION_BLOCK FB_Reactor_IO
VAR_IN_OUT
	fan_vfd																: REAL;
	inlet_co2_pump														: BOOL;
	inlet_co2_sol														: BOOL;
	outlet_co2_pump														: BOOL;
	outlet_co2_sol														: BOOL;
	repres_valve														: BOOL;
	inlet_door_clamps_extend											: BOOL;
	outlet_door_clamps_extend											: BOOL;
	inlet_door_clamps_retract											: BOOL;
	outlet_door_clamps_retract											: BOOL;
	inlet_door_open														: BOOL;
	inlet_door_close													: BOOL;
	outlet_door_open													: BOOL;
	outlet_door_close													: BOOL;
	fan_vfd_reset														: BOOL;
END_VAR
VAR_INPUT
	RSet																: STRING;
	React																: STRING;
	Power_On															: BOOL;
	
	TT_01_01															: INT;
	TT_01_01_offset														: REAL;
	TT_01_01_error														: BOOL;
	TT_01_03															: INT;
	TT_01_03_offset														: REAL;
	TT_01_03_error														: BOOL;
	TT_02_01															: INT;
	TT_02_01_offset														: REAL;
	TT_02_01_error														: BOOL;
	TT_02_03															: INT;
	TT_02_03_offset														: REAL;
	TT_02_03_error														: BOOL;
	TT_03_01															: INT;
	TT_03_01_offset														: REAL;
	TT_03_01_error														: BOOL;
	TT_03_03															: INT;
	TT_03_03_offset														: REAL;
	TT_03_03_error														: BOOL;
	TT_04_01															: INT;
	TT_04_01_offset														: REAL;
	TT_04_01_error														: BOOL;
	TT_04_03															: INT;
	TT_04_03_offset														: REAL;
	TT_04_03_error														: BOOL;
	TT_05_01															: INT;
	TT_05_01_offset														: REAL;
	TT_05_01_error														: BOOL;
	TT_05_03															: INT;
	TT_05_03_offset														: REAL;
	TT_05_03_error														: BOOL;
	TT_06_01															: INT;
	TT_06_01_offset														: REAL;
	TT_06_01_error														: BOOL;
	TT_06_03															: INT;
	TT_06_03_offset														: REAL;
	TT_06_03_error														: BOOL;
	TT_07_01															: INT;
	TT_07_01_offset														: REAL;
	TT_07_01_error														: BOOL;
	TT_07_03															: INT;
	TT_07_03_offset														: REAL;
	TT_07_03_error														: BOOL;
	TT_08_01															: INT;
	TT_08_01_offset														: REAL;
	TT_08_01_error														: BOOL;
	TT_08_03															: INT;
	TT_08_03_offset														: REAL;
	TT_08_03_error														: BOOL;
	TT_09_01															: INT;
	TT_09_01_offset														: REAL;
	TT_09_01_error														: BOOL;
	TT_09_03															: INT;
	TT_09_03_offset														: REAL;
	TT_09_03_error														: BOOL;
	TT_10_01															: INT;
	TT_10_01_offset														: REAL;
	TT_10_01_error														: BOOL;
	TT_10_03															: INT;
	TT_10_03_offset														: REAL;
	TT_10_03_error														: BOOL;
	TT_11_01															: INT;
	TT_11_01_offset														: REAL;
	TT_11_01_error														: BOOL;
	TT_11_03															: INT;
	TT_11_03_offset														: REAL;
	TT_11_03_error														: BOOL;
	TT_12_01															: INT;
	TT_12_01_offset														: REAL;
	TT_12_01_error														: BOOL;
	TT_12_03															: INT;
	TT_12_03_offset														: REAL;
	TT_12_03_error														: BOOL;
	
	bRepresValve														: BOOL;
	repres_valve_open													: BOOL;
	repres_valve_closed													: BOOL;
	
	fan_vfd_status														: WORD;
	fan_vfd_velocity													: WORD;
	fan_vfd_input														: REAL;
	fan_vfd_enable														: BOOL;
	fan_vfd_ecat_state													: BOOL;
	fan_vfd_current														: DINT;
	fan_vfd_temp														: INT;
	
	inlet_door_left_clamps_extended		 								: BOOL;
	inlet_door_right_clamps_extended	 								: BOOL;
	outlet_door_left_clamps_extended	 								: BOOL;
	outlet_door_right_clamps_extended									: BOOL;
	extend_clamps														: BOOL;
	retract_clamps														: BOOL;
	
	inlet_door_left_open												: BOOL;
	inlet_door_right_open												: BOOL;
	outlet_door_left_open												: BOOL;
	outlet_door_right_open												: BOOL;
	inlet_door_left_closed												: BOOL;
	inlet_door_right_closed												: BOOL;
	outlet_door_left_closed												: BOOL;
	outlet_door_right_closed											: BOOL;
	open_doors															: BOOL;
	close_doors															: BOOL;
	
	co2_sensor_config													: INT;
END_VAR
VAR_OUTPUT
	AT_01_pump															: BOOL;
	inlet_co2_pump_cmd_status											: BOOL;
	AT_01_sol															: BOOL;
	inlet_co2_sol_cmd_status											: BOOL;
	AT_03_pump															: BOOL;
	outlet_co2_pump_cmd_status											: BOOL;
	AT_03_sol															: BOOL;
	outlet_co2_sol_cmd_status											: BOOL;
	XV_02																: BOOL;
	repres_valve_open_cmd_status										: BOOL;
	repres_valve_clear													: BOOL;

	reactor_wall_temp													: REAL;
	reactor_wall_temp_error												: BOOL;
	outlet_line_temp													: REAL;
	outlet_line_temp_error												: BOOL;
	
	cart01_front_temp													: REAL;						
	cart01_front_temp_error 											: BOOL;
	cart01_back_temp													: REAL;
	cart01_back_temp_error 												: BOOL;
	cart02_front_temp													: REAL;						
	cart02_front_temp_error 											: BOOL;
	cart02_back_temp													: REAL;
	cart02_back_temp_error 												: BOOL;
	cart03_front_temp													: REAL;						
	cart03_front_temp_error 											: BOOL;
	cart03_back_temp													: REAL;
	cart03_back_temp_error 												: BOOL;
	cart04_front_temp													: REAL;						
	cart04_front_temp_error 											: BOOL;
	cart04_back_temp													: REAL;
	cart04_back_temp_error 												: BOOL;
	cart05_front_temp													: REAL;						
	cart05_front_temp_error 											: BOOL;
	cart05_back_temp													: REAL;
	cart05_back_temp_error 												: BOOL;
	cart06_front_temp													: REAL;						
	cart06_front_temp_error 											: BOOL;
	cart06_back_temp													: REAL;
	cart06_back_temp_error 												: BOOL;
	cart07_front_temp													: REAL;						
	cart07_front_temp_error 											: BOOL;
	cart07_back_temp													: REAL;
	cart07_back_temp_error 												: BOOL;
	cart08_front_temp													: REAL;						
	cart08_front_temp_error 											: BOOL;
	cart08_back_temp													: REAL;
	cart08_back_temp_error 												: BOOL;
	cart09_front_temp													: REAL;						
	cart09_front_temp_error 											: BOOL;
	cart09_back_temp													: REAL;
	cart09_back_temp_error 												: BOOL;
	cart10_front_temp													: REAL;						
	cart10_front_temp_error 											: BOOL;
	cart10_back_temp													: REAL;
	cart10_back_temp_error 												: BOOL;
	cart11_front_temp													: REAL;						
	cart11_front_temp_error 											: BOOL;
	cart11_back_temp													: REAL;
	cart11_back_temp_error 												: BOOL;
	cart12_front_temp													: REAL;						
	cart12_front_temp_error 											: BOOL;
	cart12_back_temp													: REAL;
	cart12_back_temp_error 												: BOOL;
	
	sorbent_low_temp													: REAL;
	sorbent_high_temp													: REAL;
	sorbent_average_temp												: REAL;

	fan_vfd_control														: WORD;
	fan_vfd_target_vel													: WORD;
	fan_vfd_enabled														: BOOL;
	fan_vfd_error														: BOOL;
	fan_vfd_output														: REAL;
	fan_vfd_current_amps												: REAL;
	fan_vfd_temp_degC													: REAL;
	
	vacuum_cooling_high_temp_count										: INT;
	adsorption_high_temp_count											: INT;
	desorption_high_temp_count											: INT;
	
	inlet_door_left_clamps_extend										: BOOL;
	inlet_door_right_clamps_extend										: BOOL;
	outlet_door_left_clamps_extend										: BOOL;
	outlet_door_right_clamps_extend										: BOOL;
	inlet_door_left_clamps_retract										: BOOL;
	inlet_door_right_clamps_retract										: BOOL;
	outlet_door_left_clamps_retract										: BOOL;
	outlet_door_right_clamps_retract									: BOOL;

	inlet_doors_clamps_extended											: BOOL;
	outlet_doors_clamps_extended										: BOOL;
	inlet_doors_clamps_retracted										: BOOL;
	outlet_doors_clamps_retracted										: BOOL;
	door_clamps_extended												: BOOL;
	door_clamps_retracted												: BOOL;
	
	open_inlet_door														: BOOL;
	close_inlet_door													: BOOL;
	open_outlet_door													: BOOL;
	close_outlet_door													: BOOL;
	doors_open															: BOOL;
	doors_closed														: BOOL;
	
END_VAR
VAR
	iNo																	: INT		:= 1;
	sRSR																: STRING;
	
	fb_Repres_Valve														: FB_Digital_Out();
	fb_Fan_Vfd_Input													: FB_Analog_Out();
	fb_Fan																: FB_VFD();

	rtrigCo2															: R_TRIG;
	iCo2Old																: INT;
	
	tonFan																: TON;
	rRpm																: REAL;
	rRpmOld																: REAL		:= 0;

	rtrigSorbentErrorCheck												: R_TRIG;
	i																	: INT;
	iCount																: ARRAY [0..23] OF INT;

	iInletAirSetpoint													: INT	:= 0;
	iTempCount															: INT;
	iHighTempCount														: INT;
	rTempTotal															: REAL;
	rTempSP																: REAL;
	rMin																: REAL;
	rMax																: REAL;
	bInterlock															: BOOL;
	
	cart01_temp_front_calc												: FB_Temperature;
	cart01_temp_back_calc												: FB_Temperature;
	cart02_temp_front_calc												: FB_Temperature;
	cart02_temp_back_calc												: FB_Temperature;
	cart03_temp_front_calc												: FB_Temperature;
	cart03_temp_back_calc												: FB_Temperature;
	cart04_temp_front_calc												: FB_Temperature;
	cart04_temp_back_calc												: FB_Temperature;
	cart05_temp_front_calc												: FB_Temperature;
	cart05_temp_back_calc												: FB_Temperature;
	cart06_temp_front_calc												: FB_Temperature;
	cart06_temp_back_calc												: FB_Temperature;
	cart07_temp_front_calc												: FB_Temperature;
	cart07_temp_back_calc												: FB_Temperature;
	cart08_temp_front_calc												: FB_Temperature;
	cart08_temp_back_calc												: FB_Temperature;
	cart09_temp_front_calc												: FB_Temperature;
	cart09_temp_back_calc												: FB_Temperature;
	cart10_temp_front_calc												: FB_Temperature;
	cart10_temp_back_calc												: FB_Temperature;
	cart11_temp_front_calc												: FB_Temperature;
	cart11_temp_back_calc												: FB_Temperature;
	cart12_temp_front_calc												: FB_Temperature;
	cart12_temp_back_calc												: FB_Temperature;
	
END_VAR

// Phase 0 - FB_Reactor_IO
// Rev 1.0 - April 26, 2024

sRSR																	:= CONCAT(RSet, React);

// CO2 SENSOR HANDLING - Tested 4/1/24
rtrigCo2(CLK:= co2_sensor_config <> iCo2Old);
IF rtrigCo2.Q THEN
	iCo2Old																:= co2_sensor_config;
	IF co2_sensor_config = 1 THEN
		inlet_co2_pump													:= TRUE;
		inlet_co2_sol													:= TRUE;
		outlet_co2_pump													:= TRUE;
		outlet_co2_sol													:= TRUE;
	ELSIF co2_sensor_config = 2 THEN
		inlet_co2_pump													:= TRUE;
		inlet_co2_sol													:= FALSE;
		outlet_co2_pump													:= TRUE;
		outlet_co2_sol													:= FALSE;
	ELSE
		inlet_co2_pump													:= FALSE;
		inlet_co2_sol													:= FALSE;
		outlet_co2_pump													:= FALSE;
		outlet_co2_sol													:= FALSE;
	END_IF
END_IF

// OUTPUTS
AT_01_pump																:= inlet_co2_pump;
inlet_co2_pump_cmd_status												:= inlet_co2_pump;

AT_01_sol																:= inlet_co2_sol;
inlet_co2_sol_cmd_status												:= inlet_co2_sol;

AT_03_pump																:= outlet_co2_pump;
outlet_co2_pump_cmd_status												:= outlet_co2_pump;

AT_03_sol																:= outlet_co2_sol;
outlet_co2_sol_cmd_status												:= outlet_co2_sol;

fb_Repres_Valve(Input1:= repres_valve, Input2:= bRepresValve, Output=> XV_02);
repres_valve_open_cmd_status											:= bRepresValve;
repres_valve_clear														:= (bRepresValve AND repres_valve_open) OR (NOT bRepresValve AND repres_valve_closed);

// SORBENT TEMPERATURE HANDLING
rtrigSorbentErrorCheck(CLK:= MAIN.bHalfSecondPulse);
IF rtrigSorbentErrorCheck.Q THEN
	A_Sorbent_Temperatures();
END_IF

// FAN
fb_Fan_Vfd_Input(Input1:= fan_vfd, Input2:= fan_vfd_input);
tonFan(IN:= fan_vfd <> rRpmOld, PT:= INT_TO_TIME((iNo - 1) * _FAN_DELAY_TIME));
IF tonFan.Q THEN
	rRpmOld																:= fan_vfd;
	rRpm																:= fan_vfd * _FAN_RPM_FACTOR;
END_IF
fb_Fan(	Enable_Vfd														:= NOT fan_vfd_ecat_state AND fan_vfd_enable,
		Fault_Reset														:= fan_vfd_reset, 
		Rpm																:= rRpm, 
		Minimum_Speed													:= _FAN_SPEED_MIN,
		Maximum_Speed													:= _FAN_SPEED_MAX, 
		StatusWord														:= fan_vfd_status, 
		ControlWord														=> fan_vfd_control, 
		TargetRpm														=> fan_vfd_target_vel, 
		Ready															=> fan_vfd_enabled,
		Error															=> fan_vfd_error);
fan_vfd_output															:= WORD_TO_REAL(fan_vfd_velocity) / _FAN_RPM_FACTOR;
fan_vfd_current_amps													:= DINT_TO_REAL(fan_vfd_current)/100;
fan_vfd_temp_degC														:= INT_TO_REAL(fan_vfd_temp);
IF fan_vfd_reset THEN
	fan_vfd_reset														:= FALSE;
END_IF

// DOORS & CLAMPS
doors_open																:= inlet_door_left_open AND inlet_door_right_open AND outlet_door_left_open AND outlet_door_right_open;
doors_closed															:= inlet_door_left_closed AND inlet_door_right_closed AND outlet_door_left_closed AND outlet_door_right_closed;

inlet_doors_clamps_extended												:= inlet_door_left_clamps_extended AND inlet_door_right_clamps_extended;
outlet_doors_clamps_extended											:= outlet_door_left_clamps_extended AND outlet_door_right_clamps_extended;	
inlet_doors_clamps_retracted											:= NOT inlet_door_left_clamps_extended AND NOT inlet_door_right_clamps_extended;
outlet_doors_clamps_retracted											:= NOT outlet_door_left_clamps_extended AND NOT outlet_door_right_clamps_extended;	
door_clamps_extended													:= inlet_doors_clamps_extended AND outlet_doors_clamps_extended;
door_clamps_retracted													:= NOT inlet_doors_clamps_extended AND NOT outlet_doors_clamps_extended;

IF inlet_door_open OR open_doors THEN
	bInterlock															:= inlet_doors_clamps_retracted;
	close_inlet_door													:= NOT bInterlock;
	open_inlet_door														:= bInterlock;
	inlet_door_open														:= FALSE;
ELSIF inlet_door_close OR close_doors THEN
	bInterlock															:= inlet_doors_clamps_retracted;
	open_inlet_door														:= NOT bInterlock;
	close_inlet_door													:= bInterlock;
	inlet_door_close													:= FALSE;
END_IF
IF outlet_door_open OR open_doors THEN
	bInterlock															:=  outlet_doors_clamps_retracted;
	close_outlet_door													:= NOT bInterlock;
	open_outlet_door													:= bInterlock;
	outlet_door_open													:= FALSE;
ELSIF outlet_door_close OR close_doors THEN
	bInterlock															:= outlet_doors_clamps_retracted;
	open_outlet_door													:= NOT bInterlock;
	close_outlet_door													:= bInterlock;
	outlet_door_close													:= FALSE;
END_IF

// CLAMPS
IF inlet_door_clamps_extend OR extend_clamps THEN
	bInterlock															:=  TRUE ; // inlet_door_left_closed AND inlet_door_right_closed;
//	bInterlock															:=  inlet_door_left_closed AND inlet_door_right_closed;
	inlet_door_left_clamps_retract										:= NOT bInterlock;
	inlet_door_right_clamps_retract										:= NOT bInterlock;
	inlet_door_left_clamps_extend										:= bInterlock;
	inlet_door_right_clamps_extend										:= bInterlock;
	inlet_door_clamps_extend											:= FALSE;
ELSIF inlet_door_clamps_retract OR retract_clamps THEN
	inlet_door_left_clamps_extend										:= FALSE;
	inlet_door_right_clamps_extend										:= FALSE;
	inlet_door_left_clamps_retract										:= TRUE;
	inlet_door_right_clamps_retract										:= TRUE;
	inlet_door_clamps_retract											:= FALSE;
END_IF
IF outlet_door_clamps_extend OR extend_clamps THEN
	bInterlock															:= TRUE ; // outlet_door_left_closed AND outlet_door_right_closed;
//	bInterlock															:= outlet_door_left_closed AND outlet_door_right_closed;
	outlet_door_left_clamps_retract										:= NOT bInterlock;
	outlet_door_right_clamps_retract									:= NOT bInterlock;
	outlet_door_left_clamps_extend										:= bInterlock;
	outlet_door_right_clamps_extend										:= bInterlock;
	outlet_door_clamps_extend											:= FALSE;
ELSIF outlet_door_clamps_retract or retract_clamps THEN
	outlet_door_left_clamps_extend										:= FALSE;
	outlet_door_right_clamps_extend										:= FALSE;
	outlet_door_left_clamps_retract										:= TRUE;
	outlet_door_right_clamps_retract									:= TRUE;
	outlet_door_clamps_retract											:= FALSE;
END_IF

ACTION A_Sorbent_Temperatures:
// Phase 0 - FB_ReatorIO.A_Sorbent_Temperatures
// Rev 1.0 - April 25, 2024

sorbent_low_temp																:= 1000;
sorbent_high_temp																:= -1000;

rTempTotal																:= 0;
iTempCount																:= 0;

cart01_front_temp														:= F_Temperature(TT_01_01, TT_01_01_offset);
cart01_front_temp_error 												:= TT_01_01_error OR iCount[0] < 30;
cart01_back_temp														:= F_Temperature(TT_01_03, TT_01_03_offset);
cart01_back_temp_error 													:= TT_01_03_Error OR iCount[1] < 30;
cart01_temp_front_calc(Error:= TT_01_01_error, Temp:= cart01_front_temp, Low:= sorbent_low_temp, High:= sorbent_high_temp, Total:= rTempTotal, Counter:= iTempCount);
cart01_temp_back_calc(Error:= TT_01_03_Error, Temp:= cart01_back_temp, Low:= sorbent_low_temp, High:= sorbent_high_temp, Total:= rTempTotal, Counter:= iTempCount);

cart02_front_temp														:= F_Temperature(TT_02_01, TT_02_01_offset);
cart02_front_temp_error 												:= TT_02_01_error OR iCount[2] < 30;
cart02_back_temp														:= F_Temperature(TT_02_03, TT_02_03_offset);
cart02_back_temp_error 													:= TT_02_03_Error OR iCount[3] < 30;
cart02_temp_front_calc(Error:= TT_02_01_error, Temp:= cart02_front_temp, Low:= sorbent_low_temp, High:= sorbent_high_temp, Total:= rTempTotal, Counter:= iTempCount);
cart02_temp_back_calc(Error:= TT_02_03_Error, Temp:= cart02_back_temp, Low:= sorbent_low_temp, High:= sorbent_high_temp, Total:= rTempTotal, Counter:= iTempCount);

cart03_front_temp														:= F_Temperature(TT_03_01, TT_03_01_offset);
cart03_front_temp_error 												:= TT_03_01_error OR iCount[4] < 30;
cart03_back_temp														:= F_Temperature(TT_03_03, TT_03_03_offset);
cart03_back_temp_error 													:= TT_03_03_Error OR iCount[5] < 30;
cart03_temp_front_calc(Error:= TT_03_01_error, Temp:= cart03_front_temp, Low:= sorbent_low_temp, High:= sorbent_high_temp, Total:= rTempTotal, Counter:= iTempCount);
cart03_temp_back_calc(Error:= TT_03_03_Error, Temp:= cart03_back_temp, Low:= sorbent_low_temp, High:= sorbent_high_temp, Total:= rTempTotal, Counter:= iTempCount);

